(* Logix 5000 project; controller reports 1756-L63 rev 20.15; software revision 20.04; part 32 of 52 *)

        [2].log_data[29].min := 1.0, [2].log_data[29].max := 1.0, [2].log_data[29].total := 3600.0, [2].log_data[29].time := 3600.0, [2].log_data[29].valid := 1, [2].log_data[30].min := 1.0, [2].log_data[30].max := 1.0, [2].log_data[30].total := 3600.0, [2].log_data[30].time := 3600.0, [2].log_data[30].valid := 1, [2].log_data[31].max := 1.0, [2].log_data[31].total := 1162.2471, [2].log_data[31].time := 3600.0, [2].log_data[31].maxminute := 16, [2].log_data[31].valid := 1, [2].log_data[32].max := 1.0, [2].log_data[32].total := 1365.247, [2].log_data[32].time := 3600.0, [2].log_data[32].maxminute := 10, [2].log_data[32].valid := 1, [2].log_data[33].time := 3600.0, [2].log_data[33].valid := 1, [2].log_data[34].time := 3600.0, [2].log_data[34].valid := 1, [2].log_data[35].max := 1.0, [2].log_data[35].total := 1525.747, [2].log_data[35].time := 3600.0, [2].log_data[35].maxminute := 10, [2].log_data[35].valid := 1, [2].log_data[36].max := 1.0, [2].log_data[36].total := 1086.749, [2].log_data[36].time := 3600.0, [2].log_data[36].maxminute := 19, [2].log_data[36].valid := 1, [2].log_data[37].max := 7.628602, [2].log_data[37].total := 3405.06, [2].log_data[37].time := 3600.0, [2].log_data[37].maxminute := 7, [2].log_data[37].valid := 1, [2].log_data[38].time := 3600.0, [2].log_data[38].valid := 1, [2].log_data[39].min := 0.9947063, [2].log_data[39].max := 1.0214411, [2].log_data[39].total := 3607.0884, [2].log_data[39].time := 3600.0, [2].log_data[39].minminute := 23, [2].log_data[39].maxminute := 9, [2].log_data[39].valid := 1, [2].log_data[40].min := 7.538759, [2].log_data[40].max := 7.5879498, [2].log_data[40].total := 27269.645, [2].log_data[40].time := 3600.0, [2].log_data[40].minminute := 15, [2].log_data[40].maxminute := 21, [2].log_data[40].valid := 1, [2].log_data[41].min := 0.046291504, [2].log_data[41].max := 0.07318335, [2].log_data[41].total := 210.1296, [2].log_data[41].time := 3600.0, [2].log_data[41].minminute := 17,
        [2].log_data[41].maxminute := 38, [2].log_data[41].valid := 1, [2].log_data[42].min := 2.2874026, [2].log_data[42].max := 2.2989445, [2].log_data[42].total := 8264.829, [2].log_data[42].time := 3600.0, [2].log_data[42].minminute := 26, [2].log_data[42].maxminute := 48, [2].log_data[42].valid := 1, [2].log_data[43].min := -0.26000214, [2].log_data[43].max := -0.26000214, [2].log_data[43].total := -935.9732, [2].log_data[43].time := 3600.0, [2].log_data[43].valid := 1, [2].log_data[44].min := -0.30000305, [2].log_data[44].max := -0.27999878, [2].log_data[44].total := -1041.974, [2].log_data[44].time := 3600.0, [2].log_data[44].valid := 1, [2].log_data[45].time := 3600.0, [2].log_data[45].valid := 1, [2].log_data[46].time := 3600.0, [2].log_data[46].valid := 1, [2].log_data[47].time := 3600.0, [2].log_data[47].valid := 1, [2].log_data[48].min := 6.583802, [2].log_data[48].max := 6.980899, [2].log_data[48].total := 24245.068, [2].log_data[48].time := 3600.0, [2].log_data[48].minminute := 38, [2].log_data[48].maxminute := 14, [2].log_data[48].valid := 1, [2].log_data[49].min := 6.739631, [2].log_data[49].max := 9.3503065, [2].log_data[49].total := 28682.559, [2].log_data[49].time := 3600.0, [2].log_data[49].minminute := 30, [2].log_data[49].maxminute := 1, [2].log_data[49].valid := 1, [2].log_data[50].min := 2.0478487, [2].log_data[50].max := 2.1506662, [2].log_data[50].total := 7513.924, [2].log_data[50].time := 3600.0, [2].log_data[50].minminute := 59, [2].log_data[50].maxminute := 10, [2].log_data[50].valid := 1, [2].log_data[51].time := 3600.0, [2].log_data[51].valid := 1, [2].log_data[52].min := -4.159996, [2].log_data[52].max := 0.11999512, [2].log_data[52].total := -7228.672, [2].log_data[52].time := 3600.0, [2].log_data[52].minminute := 10, [2].log_data[52].maxminute := 15, [2].log_data[52].valid := 1, [2].log_data[53].min := -3.899994, [2].log_data[53].max := 0.22000122, [2].log_data[53].total := -6730.6216, [2].log_data[53].time := 3600.0, [2].log_data[53].minminute := 10,
        [2].log_data[53].maxminute := 18, [2].log_data[53].valid := 1, [2].log_data[54].max := 0.519, [2].log_data[54].total := 999.3493, [2].log_data[54].time := 3600.0, [2].log_data[54].maxminute := 48, [2].log_data[54].valid := 1, [2].log_data[55].max := 0.534, [2].log_data[55].total := 1035.1941, [2].log_data[55].time := 3600.0, [2].log_data[55].maxminute := 51, [2].log_data[55].valid := 1, [2].log_data[56].min := 0.16024561, [2].log_data[56].max := 0.1607167, [2].log_data[56].total := 577.607, [2].log_data[56].time := 3600.0, [2].log_data[56].minminute := 35, [2].log_data[56].maxminute := 17, [2].log_data[56].valid := 1, [2].log_data[57].min := 0.32045865, [2].log_data[57].max := 0.3224608, [2].log_data[57].total := 1158.1218, [2].log_data[57].time := 3600.0, [2].log_data[57].minminute := 47, [2].log_data[57].maxminute := 30, [2].log_data[57].valid := 1, [2].log_data[58].time := 3600.0, [2].log_data[58].valid := 1, [2].log_data[59].time := 3600.0, [2].log_data[59].valid := 1, [2].log_data[60].valid := 1, [2].log_data[61].valid := 1, [2].log_data[62].valid := 1, [2].log_data[63].valid := 1, [2].log_data[64].valid := 1, [2].log_data[65].valid := 1, [2].log_data[66].valid := 1, [2].log_data[67].valid := 1, [2].log_data[68].valid := 1, [2].log_data[69].valid := 1, [2].log_data[70].valid := 1, [2].log_data[71].valid := 1, [2].log_data[72].valid := 1, [2].log_data[73].valid := 1, [2].log_data[74].valid := 1, [2].log_data[75].valid := 1, [2].log_data[76].valid := 1, [2].log_data[77].valid := 1, [2].log_data[78].valid := 1, [2].log_data[79].valid := 1, [2].log_data[80].valid := 1, [2].log_data[81].valid := 1, [2].log_data[82].valid := 1, [2].log_data[83].valid := 1, [2].log_data[84].valid := 1, [2].log_data[85].valid := 1, [2].log_data[86].valid := 1, [2].log_data[87].valid := 1, [2].log_data[88].valid := 1, [2].log_data[89].valid := 1,
        [2].log_data[90].valid := 1, [2].log_data[91].valid := 1, [2].log_data[92].valid := 1, [2].log_data[93].valid := 1, [2].log_data[94].valid := 1, [2].log_data[95].valid := 1, [2].log_data[96].valid := 1, [2].log_data[97].valid := 1, [2].log_data[98].valid := 1, [2].log_data[99].valid := 1, [2].log_data[100].valid := 1, [2].log_data[101].valid := 1, [2].log_data[102].valid := 1, [2].log_data[103].valid := 1, [2].log_data[104].valid := 1, [2].log_data[105].valid := 1, [2].log_data[106].valid := 1, [2].log_data[107].valid := 1, [2].log_data[108].valid := 1, [2].log_data[109].valid := 1, [2].log_data[110].valid := 1, [2].log_data[111].valid := 1, [2].log_data[112].valid := 1, [2].log_data[113].valid := 1, [2].log_data[114].valid := 1, [2].log_data[115].valid := 1, [2].log_data[116].valid := 1, [2].log_data[117].valid := 1, [2].log_data[118].valid := 1, [2].log_data[119].valid := 1, [2].log_data[120].valid := 1, [2].log_data[121].valid := 1, [2].log_data[122].valid := 1, [2].log_data[123].valid := 1, [2].log_data[124].valid := 1, [2].time.Year := 2023, [2].time.Month := 1, [2].time.Day := 13, [2].time.Hour := 5, [2].time.Minute := 59, [2].time.Second := 59, [3].log_data[0].min := 1.0, [3].log_data[0].max := 1.0, [3].log_data[0].total := 3600.0, [3].log_data[0].time := 3600.0, [3].log_data[0].valid := 1, [3].log_data[1].time := 3600.0, [3].log_data[1].valid := 1, [3].log_data[2].time := 3600.0, [3].log_data[2].valid := 1, [3].log_data[3].time := 3600.0, [3].log_data[3].valid := 1, [3].log_data[4].time := 3600.0, [3].log_data[4].valid := 1, [3].log_data[5].time := 3600.0, [3].log_data[5].valid := 1, [3].log_data[6].time := 3600.0, [3].log_data[6].valid := 1, [3].log_data[7].time := 3600.0, [3].log_data[7].valid := 1,
        [3].log_data[8].max := 1.0, [3].log_data[8].total := 2110.251, [3].log_data[8].time := 3600.0, [3].log_data[8].minminute := 35, [3].log_data[8].valid := 1, [3].log_data[9].max := 1.0, [3].log_data[9].total := 2110.251, [3].log_data[9].time := 3600.0, [3].log_data[9].minminute := 35, [3].log_data[9].valid := 1, [3].log_data[10].min := 1.0, [3].log_data[10].max := 1.0, [3].log_data[10].total := 3600.0, [3].log_data[10].time := 3600.0, [3].log_data[10].valid := 1, [3].log_data[11].time := 3600.0, [3].log_data[11].valid := 1, [3].log_data[12].min := 1.0, [3].log_data[12].max := 1.0, [3].log_data[12].total := 3600.0, [3].log_data[12].time := 3600.0, [3].log_data[12].valid := 1, [3].log_data[13].min := 1.0, [3].log_data[13].max := 1.0, [3].log_data[13].total := 3600.0, [3].log_data[13].time := 3600.0, [3].log_data[13].valid := 1, [3].log_data[14].time := 3600.0, [3].log_data[14].valid := 1, [3].log_data[15].time := 3600.0, [3].log_data[15].valid := 1, [3].log_data[16].time := 3600.0, [3].log_data[16].valid := 1, [3].log_data[17].min := 1.0, [3].log_data[17].max := 1.0, [3].log_data[17].total := 3600.0, [3].log_data[17].time := 3600.0, [3].log_data[17].valid := 1, [3].log_data[18].time := 3600.0, [3].log_data[18].valid := 1, [3].log_data[19].time := 3600.0, [3].log_data[19].valid := 1, [3].log_data[20].time := 3600.0, [3].log_data[20].valid := 1, [3].log_data[21].min := 1.0, [3].log_data[21].max := 1.0, [3].log_data[21].total := 3600.0, [3].log_data[21].time := 3600.0, [3].log_data[21].valid := 1, [3].log_data[22].time := 3600.0, [3].log_data[22].valid := 1, [3].log_data[23].time := 3600.0, [3].log_data[23].valid := 1, [3].log_data[24].time := 3600.0, [3].log_data[24].valid := 1, [3].log_data[25].time := 3600.0, [3].log_data[25].valid := 1, [3].log_data[26].time := 3600.0, [3].log_data[26].valid := 1, [3].log_data[27].time := 3600.0,
        [3].log_data[27].valid := 1, [3].log_data[28].time := 3600.0, [3].log_data[28].valid := 1, [3].log_data[29].min := 1.0, [3].log_data[29].max := 1.0, [3].log_data[29].total := 3600.0, [3].log_data[29].time := 3600.0, [3].log_data[29].valid := 1, [3].log_data[30].min := 1.0, [3].log_data[30].max := 1.0, [3].log_data[30].total := 3600.0, [3].log_data[30].time := 3600.0, [3].log_data[30].valid := 1, [3].log_data[31].max := 1.0, [3].log_data[31].total := 1010.749, [3].log_data[31].time := 3600.0, [3].log_data[31].minminute := 7, [3].log_data[31].valid := 1, [3].log_data[32].max := 1.0, [3].log_data[32].total := 838.749, [3].log_data[32].time := 3600.0, [3].log_data[32].maxminute := 9, [3].log_data[32].valid := 1, [3].log_data[33].time := 3600.0, [3].log_data[33].valid := 1, [3].log_data[34].time := 3600.0, [3].log_data[34].valid := 1, [3].log_data[35].max := 1.0, [3].log_data[35].total := 674.249, [3].log_data[35].time := 3600.0, [3].log_data[35].valid := 1, [3].log_data[36].max := 1.0, [3].log_data[36].total := 1086.498, [3].log_data[36].time := 3600.0, [3].log_data[36].maxminute := 1, [3].log_data[36].valid := 1, [3].log_data[37].time := 3600.0, [3].log_data[37].valid := 1, [3].log_data[38].time := 3600.0, [3].log_data[38].valid := 1, [3].log_data[39].min := 0.99435294, [3].log_data[39].max := 1.0062482, [3].log_data[39].total := 3601.9426, [3].log_data[39].time := 3600.0, [3].log_data[39].minminute := 6, [3].log_data[39].maxminute := 44, [3].log_data[39].valid := 1, [3].log_data[40].min := 7.5588202, [3].log_data[40].max := 7.5808053, [3].log_data[40].total := 27270.088, [3].log_data[40].time := 3600.0, [3].log_data[40].minminute := 56, [3].log_data[40].maxminute := 26, [3].log_data[40].valid := 1, [3].log_data[41].min := 0.041187745, [3].log_data[41].max := 0.071024165, [3].log_data[41].total := 188.56963, [3].log_data[41].time := 3600.0, [3].log_data[41].minminute := 21, [3].log_data[41].maxminute := 43,
        [3].log_data[41].valid := 1, [3].log_data[42].min := 2.2922316, [3].log_data[42].max := 2.3007112, [3].log_data[42].total := 8264.858, [3].log_data[42].time := 3600.0, [3].log_data[42].minminute := 23, [3].log_data[42].maxminute := 24, [3].log_data[42].valid := 1, [3].log_data[43].min := -0.26000214, [3].log_data[43].max := -0.26000214, [3].log_data[43].total := -935.9732, [3].log_data[43].time := 3600.0, [3].log_data[43].valid := 1, [3].log_data[44].min := -0.30000305, [3].log_data[44].max := -0.27999878, [3].log_data[44].total := -1052.0194, [3].log_data[44].time := 3600.0, [3].log_data[44].valid := 1, [3].log_data[45].time := 3600.0, [3].log_data[45].valid := 1, [3].log_data[46].time := 3600.0, [3].log_data[46].valid := 1, [3].log_data[47].time := 3600.0, [3].log_data[47].valid := 1, [3].log_data[48].min := 6.737969, [3].log_data[48].max := 6.778366, [3].log_data[48].total := 24290.475, [3].log_data[48].time := 3600.0, [3].log_data[48].minminute := 40, [3].log_data[48].valid := 1, [3].log_data[49].min := 8.845053, [3].log_data[49].max := 9.3279295, [3].log_data[49].total := 33251.055, [3].log_data[49].time := 3600.0, [3].log_data[49].maxminute := 42, [3].log_data[49].valid := 1, [3].log_data[50].min := 1.9994433, [3].log_data[50].max := 2.1072073, [3].log_data[50].total := 7396.8003, [3].log_data[50].time := 3600.0, [3].log_data[50].minminute := 35, [3].log_data[50].maxminute := 58, [3].log_data[50].valid := 1, [3].log_data[51].time := 3600.0, [3].log_data[51].valid := 1, [3].log_data[52].min := -2.9000015, [3].log_data[52].max := 0.11999512, [3].log_data[52].total := -6534.5815, [3].log_data[52].time := 3600.0, [3].log_data[52].minminute := 19, [3].log_data[52].maxminute := 7, [3].log_data[52].valid := 1, [3].log_data[53].min := -2.4400024, [3].log_data[53].max := 0.19999695, [3].log_data[53].total := -5788.244, [3].log_data[53].time := 3600.0, [3].log_data[53].minminute := 14, [3].log_data[53].valid := 1, [3].log_data[54].max := 0.539, [3].log_data[54].total := 734.8154,
        [3].log_data[54].time := 3600.0, [3].log_data[54].minminute := 7, [3].log_data[54].maxminute := 19, [3].log_data[54].valid := 1, [3].log_data[55].max := 0.5075, [3].log_data[55].total := 697.1523, [3].log_data[55].time := 3600.0, [3].log_data[55].maxminute := 22, [3].log_data[55].valid := 1, [3].log_data[56].min := 0.16032413, [3].log_data[56].max := 0.1607167, [3].log_data[56].total := 577.6799, [3].log_data[56].time := 3600.0, [3].log_data[56].minminute := 9, [3].log_data[56].maxminute := 2, [3].log_data[56].valid := 1, [3].log_data[57].min := 0.32045865, [3].log_data[57].max := 0.3208905, [3].log_data[57].total := 1154.3016, [3].log_data[57].time := 3600.0, [3].log_data[57].minminute := 43, [3].log_data[57].maxminute := 5, [3].log_data[57].valid := 1, [3].log_data[58].time := 3600.0, [3].log_data[58].valid := 1, [3].log_data[59].time := 3600.0, [3].log_data[59].valid := 1, [3].log_data[60].valid := 1, [3].log_data[61].valid := 1, [3].log_data[62].valid := 1, [3].log_data[63].valid := 1, [3].log_data[64].valid := 1, [3].log_data[65].valid := 1, [3].log_data[66].valid := 1, [3].log_data[67].valid := 1, [3].log_data[68].valid := 1, [3].log_data[69].valid := 1, [3].log_data[70].valid := 1, [3].log_data[71].valid := 1, [3].log_data[72].valid := 1, [3].log_data[73].valid := 1, [3].log_data[74].valid := 1, [3].log_data[75].valid := 1, [3].log_data[76].valid := 1, [3].log_data[77].valid := 1, [3].log_data[78].valid := 1, [3].log_data[79].valid := 1, [3].log_data[80].valid := 1, [3].log_data[81].valid := 1, [3].log_data[82].valid := 1, [3].log_data[83].valid := 1, [3].log_data[84].valid := 1, [3].log_data[85].valid := 1, [3].log_data[86].valid := 1, [3].log_data[87].valid := 1, [3].log_data[88].valid := 1, [3].log_data[89].valid := 1, [3].log_data[90].valid := 1, [3].log_data[91].valid := 1, [3].log_data[92].valid := 1,
        [3].log_data[93].valid := 1, [3].log_data[94].valid := 1, [3].log_data[95].valid := 1, [3].log_data[96].valid := 1, [3].log_data[97].valid := 1, [3].log_data[98].valid := 1, [3].log_data[99].valid := 1, [3].log_data[100].valid := 1, [3].log_data[101].valid := 1, [3].log_data[102].valid := 1, [3].log_data[103].valid := 1, [3].log_data[104].valid := 1, [3].log_data[105].valid := 1, [3].log_data[106].valid := 1, [3].log_data[107].valid := 1, [3].log_data[108].valid := 1, [3].log_data[109].valid := 1, [3].log_data[110].valid := 1, [3].log_data[111].valid := 1, [3].log_data[112].valid := 1, [3].log_data[113].valid := 1, [3].log_data[114].valid := 1, [3].log_data[115].valid := 1, [3].log_data[116].valid := 1, [3].log_data[117].valid := 1, [3].log_data[118].valid := 1, [3].log_data[119].valid := 1, [3].log_data[120].valid := 1, [3].log_data[121].valid := 1, [3].log_data[122].valid := 1, [3].log_data[123].valid := 1, [3].log_data[124].valid := 1, [3].time.Year := 2023, [3].time.Month := 1, [3].time.Day := 13, [3].time.Hour := 6, [3].time.Minute := 59, [3].time.Second := 59, [4].log_data[0].min := 1.0, [4].log_data[0].max := 1.0, [4].log_data[0].total := 3600.0, [4].log_data[0].time := 3600.0, [4].log_data[0].valid := 1, [4].log_data[1].time := 3600.0, [4].log_data[1].valid := 1, [4].log_data[2].time := 3600.0, [4].log_data[2].valid := 1, [4].log_data[3].time := 3600.0, [4].log_data[3].valid := 1, [4].log_data[4].time := 3600.0, [4].log_data[4].valid := 1, [4].log_data[5].time := 3600.0, [4].log_data[5].valid := 1, [4].log_data[6].time := 3600.0, [4].log_data[6].valid := 1, [4].log_data[7].time := 3600.0, [4].log_data[7].valid := 1, [4].log_data[8].time := 3600.0, [4].log_data[8].valid := 1, [4].log_data[9].time := 3600.0,
        [4].log_data[9].valid := 1, [4].log_data[10].min := 1.0, [4].log_data[10].max := 1.0, [4].log_data[10].total := 3600.0, [4].log_data[10].time := 3600.0, [4].log_data[10].valid := 1, [4].log_data[11].time := 3600.0, [4].log_data[11].valid := 1, [4].log_data[12].min := 1.0, [4].log_data[12].max := 1.0, [4].log_data[12].total := 3600.0, [4].log_data[12].time := 3600.0, [4].log_data[12].valid := 1, [4].log_data[13].min := 1.0, [4].log_data[13].max := 1.0, [4].log_data[13].total := 3600.0, [4].log_data[13].time := 3600.0, [4].log_data[13].valid := 1, [4].log_data[14].time := 3600.0, [4].log_data[14].valid := 1, [4].log_data[15].time := 3600.0, [4].log_data[15].valid := 1, [4].log_data[16].time := 3600.0, [4].log_data[16].valid := 1, [4].log_data[17].min := 1.0, [4].log_data[17].max := 1.0, [4].log_data[17].total := 3600.0, [4].log_data[17].time := 3600.0, [4].log_data[17].valid := 1, [4].log_data[18].time := 3600.0, [4].log_data[18].valid := 1, [4].log_data[19].time := 3600.0, [4].log_data[19].valid := 1, [4].log_data[20].time := 3600.0, [4].log_data[20].valid := 1, [4].log_data[21].min := 1.0, [4].log_data[21].max := 1.0, [4].log_data[21].total := 3600.0, [4].log_data[21].time := 3600.0, [4].log_data[21].valid := 1, [4].log_data[22].time := 3600.0, [4].log_data[22].valid := 1, [4].log_data[23].time := 3600.0, [4].log_data[23].valid := 1, [4].log_data[24].time := 3600.0, [4].log_data[24].valid := 1, [4].log_data[25].time := 3600.0, [4].log_data[25].valid := 1, [4].log_data[26].time := 3600.0, [4].log_data[26].valid := 1, [4].log_data[27].time := 3600.0, [4].log_data[27].valid := 1, [4].log_data[28].time := 3600.0, [4].log_data[28].valid := 1, [4].log_data[29].min := 1.0, [4].log_data[29].max := 1.0, [4].log_data[29].total := 3600.0, [4].log_data[29].time := 3600.0, [4].log_data[29].valid := 1, [4].log_data[30].min := 1.0,
        [4].log_data[30].max := 1.0, [4].log_data[30].total := 3600.0, [4].log_data[30].time := 3600.0, [4].log_data[30].valid := 1, [4].log_data[31].time := 3600.0, [4].log_data[31].valid := 1, [4].log_data[32].time := 3600.0, [4].log_data[32].valid := 1, [4].log_data[33].time := 3600.0, [4].log_data[33].valid := 1, [4].log_data[34].time := 3600.0, [4].log_data[34].valid := 1, [4].log_data[35].time := 3600.0, [4].log_data[35].valid := 1, [4].log_data[36].time := 3600.0, [4].log_data[36].valid := 1, [4].log_data[37].time := 3600.0, [4].log_data[37].valid := 1, [4].log_data[38].time := 3600.0, [4].log_data[38].valid := 1, [4].log_data[39].min := 0.99423516, [4].log_data[39].max := 1.0055416, [4].log_data[39].total := 3602.0474, [4].log_data[39].time := 3600.0, [4].log_data[39].minminute := 13, [4].log_data[39].maxminute := 34, [4].log_data[39].valid := 1, [4].log_data[40].min := 7.5442557, [4].log_data[40].max := 7.5989423, [4].log_data[40].total := 27264.574, [4].log_data[40].time := 3600.0, [4].log_data[40].minminute := 22, [4].log_data[40].maxminute := 4, [4].log_data[40].valid := 1, [4].log_data[41].min := 0.0402063, [4].log_data[41].max := 0.07514624, [4].log_data[41].total := 193.19824, [4].log_data[41].time := 3600.0, [4].log_data[41].minminute := 58, [4].log_data[41].maxminute := 6, [4].log_data[41].valid := 1, [4].log_data[42].min := 2.2928205, [4].log_data[42].max := 2.298827, [4].log_data[42].total := 8264.684, [4].log_data[42].time := 3600.0, [4].log_data[42].minminute := 17, [4].log_data[42].maxminute := 44, [4].log_data[42].valid := 1, [4].log_data[43].min := -0.26000214, [4].log_data[43].max := -0.26000214, [4].log_data[43].total := -935.9732, [4].log_data[43].time := 3600.0, [4].log_data[43].valid := 1, [4].log_data[44].min := -0.30000305, [4].log_data[44].max := -0.27999878, [4].log_data[44].total := -1033.2828, [4].log_data[44].time := 3600.0, [4].log_data[44].valid := 1, [4].log_data[45].time := 3600.0, [4].log_data[45].valid := 1,
        [4].log_data[46].time := 3600.0, [4].log_data[46].valid := 1, [4].log_data[47].time := 3600.0, [4].log_data[47].valid := 1, [4].log_data[48].min := 6.740717, [4].log_data[48].max := 6.752809, [4].log_data[48].total := 24294.328, [4].log_data[48].time := 3600.0, [4].log_data[48].maxminute := 46, [4].log_data[48].valid := 1, [4].log_data[49].min := 9.282979, [4].log_data[49].max := 9.357571, [4].log_data[49].total := 33554.664, [4].log_data[49].time := 3600.0, [4].log_data[49].minminute := 3, [4].log_data[49].maxminute := 59, [4].log_data[49].valid := 1, [4].log_data[50].min := 2.1007297, [4].log_data[50].max := 2.111447, [4].log_data[50].total := 7586.518, [4].log_data[50].time := 3600.0, [4].log_data[50].minminute := 1, [4].log_data[50].maxminute := 28, [4].log_data[50].valid := 1, [4].log_data[51].time := 3600.0, [4].log_data[51].valid := 1, [4].log_data[52].min := -1.6200027, [4].log_data[52].max := -1.4400024, [4].log_data[52].total := -5511.6133, [4].log_data[52].time := 3600.0, [4].log_data[52].minminute := 37, [4].log_data[52].maxminute := 2, [4].log_data[52].valid := 1, [4].log_data[53].min := -1.5200043, [4].log_data[53].max := -1.340004, [4].log_data[53].total := -5191.9697, [4].log_data[53].time := 3600.0, [4].log_data[53].minminute := 27, [4].log_data[53].maxminute := 3, [4].log_data[53].valid := 1, [4].log_data[54].time := 3600.0, [4].log_data[54].valid := 1, [4].log_data[55].time := 3600.0, [4].log_data[55].valid := 1, [4].log_data[56].min := 0.16028486, [4].log_data[56].max := 0.16067745, [4].log_data[56].total := 577.60114, [4].log_data[56].time := 3600.0, [4].log_data[56].minminute := 3, [4].log_data[56].maxminute := 20, [4].log_data[56].valid := 1, [4].log_data[57].min := 0.32045865, [4].log_data[57].max := 0.32092974, [4].log_data[57].total := 1154.3279, [4].log_data[57].time := 3600.0, [4].log_data[57].minminute := 14, [4].log_data[57].maxminute := 51, [4].log_data[57].valid := 1, [4].log_data[58].time := 3600.0, [4].log_data[58].valid := 1,
        [4].log_data[59].time := 3600.0, [4].log_data[59].valid := 1, [4].log_data[60].valid := 1, [4].log_data[61].valid := 1, [4].log_data[62].valid := 1, [4].log_data[63].valid := 1, [4].log_data[64].valid := 1, [4].log_data[65].valid := 1, [4].log_data[66].valid := 1, [4].log_data[67].valid := 1, [4].log_data[68].valid := 1, [4].log_data[69].valid := 1, [4].log_data[70].valid := 1, [4].log_data[71].valid := 1, [4].log_data[72].valid := 1, [4].log_data[73].valid := 1, [4].log_data[74].valid := 1, [4].log_data[75].valid := 1, [4].log_data[76].valid := 1, [4].log_data[77].valid := 1, [4].log_data[78].valid := 1, [4].log_data[79].valid := 1, [4].log_data[80].valid := 1, [4].log_data[81].valid := 1, [4].log_data[82].valid := 1, [4].log_data[83].valid := 1, [4].log_data[84].valid := 1, [4].log_data[85].valid := 1, [4].log_data[86].valid := 1, [4].log_data[87].valid := 1, [4].log_data[88].valid := 1, [4].log_data[89].valid := 1, [4].log_data[90].valid := 1, [4].log_data[91].valid := 1, [4].log_data[92].valid := 1, [4].log_data[93].valid := 1, [4].log_data[94].valid := 1, [4].log_data[95].valid := 1, [4].log_data[96].valid := 1, [4].log_data[97].valid := 1, [4].log_data[98].valid := 1, [4].log_data[99].valid := 1, [4].log_data[100].valid := 1, [4].log_data[101].valid := 1, [4].log_data[102].valid := 1, [4].log_data[103].valid := 1, [4].log_data[104].valid := 1, [4].log_data[105].valid := 1, [4].log_data[106].valid := 1, [4].log_data[107].valid := 1, [4].log_data[108].valid := 1, [4].log_data[109].valid := 1, [4].log_data[110].valid := 1, [4].log_data[111].valid := 1, [4].log_data[112].valid := 1, [4].log_data[113].valid := 1, [4].log_data[114].valid := 1, [4].log_data[115].valid := 1, [4].log_data[116].valid := 1, [4].log_data[117].valid := 1,
        [4].log_data[118].valid := 1, [4].log_data[119].valid := 1, [4].log_data[120].valid := 1, [4].log_data[121].valid := 1, [4].log_data[122].valid := 1, [4].log_data[123].valid := 1, [4].log_data[124].valid := 1, [4].time.Year := 2023, [4].time.Month := 1, [4].time.Day := 13, [4].time.Hour := 7, [4].time.Minute := 59, [4].time.Second := 59, [5].log_data[0].min := 1.0, [5].log_data[0].max := 1.0, [5].log_data[0].total := 3600.0, [5].log_data[0].time := 3600.0, [5].log_data[0].valid := 1, [5].log_data[1].max := 1.0, [5].log_data[1].total := 575.0, [5].log_data[1].time := 3600.0, [5].log_data[1].maxminute := 33, [5].log_data[1].valid := 1, [5].log_data[2].max := 1.0, [5].log_data[2].total := 571.5, [5].log_data[2].time := 3600.0, [5].log_data[2].maxminute := 33, [5].log_data[2].valid := 1, [5].log_data[3].time := 3600.0, [5].log_data[3].valid := 1, [5].log_data[4].time := 3600.0, [5].log_data[4].valid := 1, [5].log_data[5].max := 1.0, [5].log_data[5].total := 230.0, [5].log_data[5].time := 3600.0, [5].log_data[5].maxminute := 35, [5].log_data[5].valid := 1, [5].log_data[6].time := 3600.0, [5].log_data[6].valid := 1, [5].log_data[7].time := 3600.0, [5].log_data[7].valid := 1, [5].log_data[8].max := 1.0, [5].log_data[8].total := 1354.249, [5].log_data[8].time := 3600.0, [5].log_data[8].maxminute := 37, [5].log_data[8].valid := 1, [5].log_data[9].max := 1.0, [5].log_data[9].total := 1350.749, [5].log_data[9].time := 3600.0, [5].log_data[9].maxminute := 37, [5].log_data[9].valid := 1, [5].log_data[10].min := 1.0, [5].log_data[10].max := 1.0, [5].log_data[10].total := 3600.0, [5].log_data[10].time := 3600.0, [5].log_data[10].valid := 1, [5].log_data[11].time := 3600.0, [5].log_data[11].valid := 1, [5].log_data[12].min := 1.0, [5].log_data[12].max := 1.0,
        [5].log_data[12].total := 3600.0, [5].log_data[12].time := 3600.0, [5].log_data[12].valid := 1, [5].log_data[13].min := 1.0, [5].log_data[13].max := 1.0, [5].log_data[13].total := 3600.0, [5].log_data[13].time := 3600.0, [5].log_data[13].valid := 1, [5].log_data[14].time := 3600.0, [5].log_data[14].valid := 1, [5].log_data[15].time := 3600.0, [5].log_data[15].valid := 1, [5].log_data[16].time := 3600.0, [5].log_data[16].valid := 1, [5].log_data[17].min := 1.0, [5].log_data[17].max := 1.0, [5].log_data[17].total := 3600.0, [5].log_data[17].time := 3600.0, [5].log_data[17].valid := 1, [5].log_data[18].time := 3600.0, [5].log_data[18].valid := 1, [5].log_data[19].time := 3600.0, [5].log_data[19].valid := 1, [5].log_data[20].time := 3600.0, [5].log_data[20].valid := 1, [5].log_data[21].min := 1.0, [5].log_data[21].max := 1.0, [5].log_data[21].total := 3600.0, [5].log_data[21].time := 3600.0, [5].log_data[21].valid := 1, [5].log_data[22].time := 3600.0, [5].log_data[22].valid := 1, [5].log_data[23].time := 3600.0, [5].log_data[23].valid := 1, [5].log_data[24].time := 3600.0, [5].log_data[24].valid := 1, [5].log_data[25].time := 3600.0, [5].log_data[25].valid := 1, [5].log_data[26].time := 3600.0, [5].log_data[26].valid := 1, [5].log_data[27].time := 3600.0, [5].log_data[27].valid := 1, [5].log_data[28].time := 3600.0, [5].log_data[28].valid := 1, [5].log_data[29].min := 1.0, [5].log_data[29].max := 1.0, [5].log_data[29].total := 3600.0, [5].log_data[29].time := 3600.0, [5].log_data[29].valid := 1, [5].log_data[30].min := 1.0, [5].log_data[30].max := 1.0, [5].log_data[30].total := 3600.0, [5].log_data[30].time := 3600.0, [5].log_data[30].valid := 1, [5].log_data[31].max := 1.0, [5].log_data[31].total := 627.498, [5].log_data[31].time := 3600.0, [5].log_data[31].maxminute := 37, [5].log_data[31].valid := 1, [5].log_data[32].max := 1.0,
        [5].log_data[32].total := 543.5, [5].log_data[32].time := 3600.0, [5].log_data[32].maxminute := 43, [5].log_data[32].valid := 1, [5].log_data[33].time := 3600.0, [5].log_data[33].valid := 1, [5].log_data[34].time := 3600.0, [5].log_data[34].valid := 1, [5].log_data[35].max := 1.0, [5].log_data[35].total := 543.249, [5].log_data[35].time := 3600.0, [5].log_data[35].maxminute := 46, [5].log_data[35].valid := 1, [5].log_data[36].max := 1.0, [5].log_data[36].total := 623.998, [5].log_data[36].time := 3600.0, [5].log_data[36].maxminute := 37, [5].log_data[36].valid := 1, [5].log_data[37].max := 7.016958, [5].log_data[37].total := 3500.9973, [5].log_data[37].time := 3600.0, [5].log_data[37].maxminute := 34, [5].log_data[37].valid := 1, [5].log_data[38].time := 3600.0, [5].log_data[38].valid := 1, [5].log_data[39].min := 0.9950596, [5].log_data[39].max := 1.0221478, [5].log_data[39].total := 3609.0261, [5].log_data[39].time := 3600.0, [5].log_data[39].minminute := 4, [5].log_data[39].maxminute := 41, [5].log_data[39].valid := 1, [5].log_data[40].min := 7.5459046, [5].log_data[40].max := 7.590698, [5].log_data[40].total := 27268.496, [5].log_data[40].time := 3600.0, [5].log_data[40].minminute := 59, [5].log_data[40].maxminute := 18, [5].log_data[40].valid := 1, [5].log_data[41].min := 0.030980714, [5].log_data[41].max := 0.058854003, [5].log_data[41].total := 181.6538, [5].log_data[41].time := 3600.0, [5].log_data[41].minminute := 21, [5].log_data[41].maxminute := 15, [5].log_data[41].valid := 1, [5].log_data[42].min := 2.2922316, [5].log_data[42].max := 2.2984736, [5].log_data[42].total := 8264.53, [5].log_data[42].time := 3600.0, [5].log_data[42].minminute := 44, [5].log_data[42].maxminute := 32, [5].log_data[42].valid := 1, [5].log_data[43].min := -0.26000214, [5].log_data[43].max := -0.26000214, [5].log_data[43].total := -935.9732, [5].log_data[43].time := 3600.0, [5].log_data[43].valid := 1, [5].log_data[44].min := -0.30000305, [5].log_data[44].max := -0.27999878,
        [5].log_data[44].total := -1029.0885, [5].log_data[44].time := 3600.0, [5].log_data[44].valid := 1, [5].log_data[45].time := 3600.0, [5].log_data[45].valid := 1, [5].log_data[46].time := 3600.0, [5].log_data[46].valid := 1, [5].log_data[47].time := 3600.0, [5].log_data[47].valid := 1, [5].log_data[48].min := 6.6137557, [5].log_data[48].max := 6.9366555, [5].log_data[48].total := 24325.88, [5].log_data[48].time := 3600.0, [5].log_data[48].minminute := 59, [5].log_data[48].maxminute := 38, [5].log_data[48].valid := 1, [5].log_data[49].min := 6.740613, [5].log_data[49].max := 9.397221, [5].log_data[49].total := 31461.621, [5].log_data[49].time := 3600.0, [5].log_data[49].minminute := 59, [5].log_data[49].maxminute := 24, [5].log_data[49].valid := 1, [5].log_data[50].min := 2.0649261, [5].log_data[50].max := 2.1504307, [5].log_data[50].total := 7575.8022, [5].log_data[50].time := 3600.0, [5].log_data[50].minminute := 41, [5].log_data[50].maxminute := 37, [5].log_data[50].valid := 1, [5].log_data[51].time := 3600.0, [5].log_data[51].valid := 1, [5].log_data[52].min := -4.199997, [5].log_data[52].max := 0.11999512, [5].log_data[52].total := -6420.016, [5].log_data[52].time := 3600.0, [5].log_data[52].minminute := 37, [5].log_data[52].maxminute := 41, [5].log_data[52].valid := 1, [5].log_data[53].min := -3.9399948, [5].log_data[53].max := 0.22000122, [5].log_data[53].total := -5998.357, [5].log_data[53].time := 3600.0, [5].log_data[53].minminute := 37, [5].log_data[53].maxminute := 45, [5].log_data[53].valid := 1, [5].log_data[54].max := 0.51199996, [5].log_data[54].total := 462.47607, [5].log_data[54].time := 3600.0, [5].log_data[54].maxminute := 53, [5].log_data[54].valid := 1, [5].log_data[55].max := 0.5145, [5].log_data[55].total := 460.84094, [5].log_data[55].time := 3600.0, [5].log_data[55].maxminute := 46, [5].log_data[55].valid := 1, [5].log_data[56].min := 0.16016708, [5].log_data[56].max := 0.1607167, [5].log_data[56].total := 577.5164, [5].log_data[56].time := 3600.0,
        [5].log_data[56].minminute := 30, [5].log_data[56].maxminute := 2, [5].log_data[56].valid := 1, [5].log_data[57].min := 0.3204979, [5].log_data[57].max := 0.32092974, [5].log_data[57].total := 1154.4246, [5].log_data[57].time := 3600.0, [5].log_data[57].minminute := 54, [5].log_data[57].maxminute := 15, [5].log_data[57].valid := 1, [5].log_data[58].time := 3600.0, [5].log_data[58].valid := 1, [5].log_data[59].time := 3600.0, [5].log_data[59].valid := 1, [5].log_data[60].valid := 1, [5].log_data[61].valid := 1, [5].log_data[62].valid := 1, [5].log_data[63].valid := 1, [5].log_data[64].valid := 1, [5].log_data[65].valid := 1, [5].log_data[66].valid := 1, [5].log_data[67].valid := 1, [5].log_data[68].valid := 1, [5].log_data[69].valid := 1, [5].log_data[70].valid := 1, [5].log_data[71].valid := 1, [5].log_data[72].valid := 1, [5].log_data[73].valid := 1, [5].log_data[74].valid := 1, [5].log_data[75].valid := 1, [5].log_data[76].valid := 1, [5].log_data[77].valid := 1, [5].log_data[78].valid := 1, [5].log_data[79].valid := 1, [5].log_data[80].valid := 1, [5].log_data[81].valid := 1, [5].log_data[82].valid := 1, [5].log_data[83].valid := 1, [5].log_data[84].valid := 1, [5].log_data[85].valid := 1, [5].log_data[86].valid := 1, [5].log_data[87].valid := 1, [5].log_data[88].valid := 1, [5].log_data[89].valid := 1, [5].log_data[90].valid := 1, [5].log_data[91].valid := 1, [5].log_data[92].valid := 1, [5].log_data[93].valid := 1, [5].log_data[94].valid := 1, [5].log_data[95].valid := 1, [5].log_data[96].valid := 1, [5].log_data[97].valid := 1, [5].log_data[98].valid := 1, [5].log_data[99].valid := 1, [5].log_data[100].valid := 1, [5].log_data[101].valid := 1, [5].log_data[102].valid := 1, [5].log_data[103].valid := 1, [5].log_data[104].valid := 1, [5].log_data[105].valid := 1,
        [5].log_data[106].valid := 1, [5].log_data[107].valid := 1, [5].log_data[108].valid := 1, [5].log_data[109].valid := 1, [5].log_data[110].valid := 1, [5].log_data[111].valid := 1, [5].log_data[112].valid := 1, [5].log_data[113].valid := 1, [5].log_data[114].valid := 1, [5].log_data[115].valid := 1, [5].log_data[116].valid := 1, [5].log_data[117].valid := 1, [5].log_data[118].valid := 1, [5].log_data[119].valid := 1, [5].log_data[120].valid := 1, [5].log_data[121].valid := 1, [5].log_data[122].valid := 1, [5].log_data[123].valid := 1, [5].log_data[124].valid := 1, [5].time.Year := 2023, [5].time.Month := 1, [5].time.Day := 13, [5].time.Hour := 8, [5].time.Minute := 59, [5].time.Second := 59, [6].log_data[0].min := 1.0, [6].log_data[0].max := 1.0, [6].log_data[0].total := 3600.0, [6].log_data[0].time := 3600.0, [6].log_data[0].valid := 1, [6].log_data[1].max := 1.0, [6].log_data[1].total := 275.249, [6].log_data[1].time := 3600.0, [6].log_data[1].maxminute := 55, [6].log_data[1].valid := 1, [6].log_data[2].max := 1.0, [6].log_data[2].total := 271.749, [6].log_data[2].time := 3600.0, [6].log_data[2].maxminute := 55, [6].log_data[2].valid := 1, [6].log_data[3].time := 3600.0, [6].log_data[3].valid := 1, [6].log_data[4].time := 3600.0, [6].log_data[4].valid := 1, [6].log_data[5].max := 1.0, [6].log_data[5].total := 125.5, [6].log_data[5].time := 3600.0, [6].log_data[5].maxminute := 57, [6].log_data[5].valid := 1, [6].log_data[6].time := 3600.0, [6].log_data[6].valid := 1, [6].log_data[7].time := 3600.0, [6].log_data[7].valid := 1, [6].log_data[8].min := 1.0, [6].log_data[8].max := 1.0, [6].log_data[8].total := 3600.0, [6].log_data[8].time := 3600.0, [6].log_data[8].valid := 1, [6].log_data[9].min := 1.0, [6].log_data[9].max := 1.0,
        [6].log_data[9].total := 3600.0, [6].log_data[9].time := 3600.0, [6].log_data[9].valid := 1, [6].log_data[10].min := 1.0, [6].log_data[10].max := 1.0, [6].log_data[10].total := 3600.0, [6].log_data[10].time := 3600.0, [6].log_data[10].valid := 1, [6].log_data[11].time := 3600.0, [6].log_data[11].valid := 1, [6].log_data[12].min := 1.0, [6].log_data[12].max := 1.0, [6].log_data[12].total := 3600.0, [6].log_data[12].time := 3600.0, [6].log_data[12].valid := 1, [6].log_data[13].min := 1.0, [6].log_data[13].max := 1.0, [6].log_data[13].total := 3600.0, [6].log_data[13].time := 3600.0, [6].log_data[13].valid := 1, [6].log_data[14].time := 3600.0, [6].log_data[14].valid := 1, [6].log_data[15].time := 3600.0, [6].log_data[15].valid := 1, [6].log_data[16].time := 3600.0, [6].log_data[16].valid := 1, [6].log_data[17].min := 1.0, [6].log_data[17].max := 1.0, [6].log_data[17].total := 3600.0, [6].log_data[17].time := 3600.0, [6].log_data[17].valid := 1, [6].log_data[18].time := 3600.0, [6].log_data[18].valid := 1, [6].log_data[19].time := 3600.0, [6].log_data[19].valid := 1, [6].log_data[20].time := 3600.0, [6].log_data[20].valid := 1, [6].log_data[21].min := 1.0, [6].log_data[21].max := 1.0, [6].log_data[21].total := 3600.0, [6].log_data[21].time := 3600.0, [6].log_data[21].valid := 1, [6].log_data[22].time := 3600.0, [6].log_data[22].valid := 1, [6].log_data[23].time := 3600.0, [6].log_data[23].valid := 1, [6].log_data[24].time := 3600.0, [6].log_data[24].valid := 1, [6].log_data[25].time := 3600.0, [6].log_data[25].valid := 1, [6].log_data[26].time := 3600.0, [6].log_data[26].valid := 1, [6].log_data[27].time := 3600.0, [6].log_data[27].valid := 1, [6].log_data[28].time := 3600.0, [6].log_data[28].valid := 1, [6].log_data[29].min := 1.0, [6].log_data[29].max := 1.0, [6].log_data[29].total := 3600.0, [6].log_data[29].time := 3600.0,
        [6].log_data[29].valid := 1, [6].log_data[30].min := 1.0, [6].log_data[30].max := 1.0, [6].log_data[30].total := 3600.0, [6].log_data[30].time := 3600.0, [6].log_data[30].valid := 1, [6].log_data[31].max := 1.0, [6].log_data[31].total := 1440.7471, [6].log_data[31].time := 3600.0, [6].log_data[31].minminute := 2, [6].log_data[31].valid := 1, [6].log_data[32].max := 1.0, [6].log_data[32].total := 1629.998, [6].log_data[32].time := 3600.0, [6].log_data[32].maxminute := 4, [6].log_data[32].valid := 1, [6].log_data[33].time := 3600.0, [6].log_data[33].valid := 1, [6].log_data[34].time := 3600.0, [6].log_data[34].valid := 1, [6].log_data[35].max := 1.0, [6].log_data[35].total := 1629.7471, [6].log_data[35].time := 3600.0, [6].log_data[35].maxminute := 7, [6].log_data[35].valid := 1, [6].log_data[36].max := 1.0, [6].log_data[36].total := 1440.7471, [6].log_data[36].time := 3600.0, [6].log_data[36].minminute := 5, [6].log_data[36].valid := 1, [6].log_data[37].max := 7.609758, [6].log_data[37].total := 2055.723, [6].log_data[37].time := 3600.0, [6].log_data[37].maxminute := 57, [6].log_data[37].valid := 1, [6].log_data[38].time := 3600.0, [6].log_data[38].valid := 1, [6].log_data[39].min := 0.99647284, [6].log_data[39].max := 1.0217944, [6].log_data[39].total := 3609.599, [6].log_data[39].time := 3600.0, [6].log_data[39].minminute := 1, [6].log_data[39].maxminute := 58, [6].log_data[39].valid := 1, [6].log_data[40].min := 7.5373855, [6].log_data[40].max := 7.591798, [6].log_data[40].total := 27273.166, [6].log_data[40].time := 3600.0, [6].log_data[40].maxminute := 6, [6].log_data[40].valid := 1, [6].log_data[41].min := 0.039028566, [6].log_data[41].max := 0.072005615, [6].log_data[41].total := 181.46281, [6].log_data[41].time := 3600.0, [6].log_data[41].minminute := 28, [6].log_data[41].maxminute := 36, [6].log_data[41].valid := 1, [6].log_data[42].min := 2.2928205, [6].log_data[42].max := 2.298827, [6].log_data[42].total := 8264.55,
        [6].log_data[42].time := 3600.0, [6].log_data[42].minminute := 2, [6].log_data[42].maxminute := 36, [6].log_data[42].valid := 1, [6].log_data[43].min := -0.27999878, [6].log_data[43].max := -0.26000214, [6].log_data[43].total := -935.9933, [6].log_data[43].time := 3600.0, [6].log_data[43].minminute := 28, [6].log_data[43].valid := 1, [6].log_data[44].min := -0.30000305, [6].log_data[44].max := -0.27999878, [6].log_data[44].total := -1067.1584, [6].log_data[44].time := 3600.0, [6].log_data[44].valid := 1, [6].log_data[45].time := 3600.0, [6].log_data[45].valid := 1, [6].log_data[46].time := 3600.0, [6].log_data[46].valid := 1, [6].log_data[47].time := 3600.0, [6].log_data[47].valid := 1, [6].log_data[48].min := 6.5821533, [6].log_data[48].max := 6.8849916, [6].log_data[48].total := 24246.365, [6].log_data[48].time := 3600.0, [6].log_data[48].minminute := 4, [6].log_data[48].maxminute := 59, [6].log_data[48].valid := 1, [6].log_data[49].min := 6.760046, [6].log_data[49].max := 9.362476, [6].log_data[49].total := 30855.816, [6].log_data[49].time := 3600.0, [6].log_data[49].maxminute := 58, [6].log_data[49].valid := 1, [6].log_data[50].min := 2.0038009, [6].log_data[50].max := 2.0876565, [6].log_data[50].total := 7366.0083, [6].log_data[50].time := 3600.0, [6].log_data[50].minminute := 57, [6].log_data[50].valid := 1, [6].log_data[51].time := 3600.0, [6].log_data[51].valid := 1, [6].log_data[52].min := -3.040001, [6].log_data[52].max := 0.11999512, [6].log_data[52].total := -7493.9536, [6].log_data[52].time := 3600.0, [6].log_data[52].minminute := 14, [6].log_data[52].maxminute := 2, [6].log_data[52].valid := 1, [6].log_data[53].min := -2.4400024, [6].log_data[53].max := 0.27999878, [6].log_data[53].total := -6821.222, [6].log_data[53].time := 3600.0, [6].log_data[53].minminute := 57, [6].log_data[53].maxminute := 6, [6].log_data[53].valid := 1, [6].log_data[54].max := 0.55550003, [6].log_data[54].total := 1217.0961, [6].log_data[54].time := 3600.0, [6].log_data[54].minminute := 2,
        [6].log_data[54].maxminute := 14, [6].log_data[54].valid := 1, [6].log_data[55].max := 0.517, [6].log_data[55].total := 1217.7288, [6].log_data[55].time := 3600.0, [6].log_data[55].minminute := 5, [6].log_data[55].maxminute := 7, [6].log_data[55].valid := 1, [6].log_data[56].min := 0.16016708, [6].log_data[56].max := 0.16067745, [6].log_data[56].total := 577.3738, [6].log_data[56].time := 3600.0, [6].log_data[56].minminute := 5, [6].log_data[56].maxminute := 34, [6].log_data[56].valid := 1, [6].log_data[57].min := 0.3184172, [6].log_data[57].max := 0.3208512, [6].log_data[57].total := 1147.9331, [6].log_data[57].time := 3600.0, [6].log_data[57].minminute := 40, [6].log_data[57].valid := 1, [6].log_data[58].time := 3600.0, [6].log_data[58].valid := 1, [6].log_data[59].time := 3600.0, [6].log_data[59].valid := 1, [6].log_data[60].valid := 1, [6].log_data[61].valid := 1, [6].log_data[62].valid := 1, [6].log_data[63].valid := 1, [6].log_data[64].valid := 1, [6].log_data[65].valid := 1, [6].log_data[66].valid := 1, [6].log_data[67].valid := 1, [6].log_data[68].valid := 1, [6].log_data[69].valid := 1, [6].log_data[70].valid := 1, [6].log_data[71].valid := 1, [6].log_data[72].valid := 1, [6].log_data[73].valid := 1, [6].log_data[74].valid := 1, [6].log_data[75].valid := 1, [6].log_data[76].valid := 1, [6].log_data[77].valid := 1, [6].log_data[78].valid := 1, [6].log_data[79].valid := 1, [6].log_data[80].valid := 1, [6].log_data[81].valid := 1, [6].log_data[82].valid := 1, [6].log_data[83].valid := 1, [6].log_data[84].valid := 1, [6].log_data[85].valid := 1, [6].log_data[86].valid := 1, [6].log_data[87].valid := 1, [6].log_data[88].valid := 1, [6].log_data[89].valid := 1, [6].log_data[90].valid := 1, [6].log_data[91].valid := 1, [6].log_data[92].valid := 1, [6].log_data[93].valid := 1, [6].log_data[94].valid := 1,
        [6].log_data[95].valid := 1, [6].log_data[96].valid := 1, [6].log_data[97].valid := 1, [6].log_data[98].valid := 1, [6].log_data[99].valid := 1, [6].log_data[100].valid := 1, [6].log_data[101].valid := 1, [6].log_data[102].valid := 1, [6].log_data[103].valid := 1, [6].log_data[104].valid := 1, [6].log_data[105].valid := 1, [6].log_data[106].valid := 1, [6].log_data[107].valid := 1, [6].log_data[108].valid := 1, [6].log_data[109].valid := 1, [6].log_data[110].valid := 1, [6].log_data[111].valid := 1, [6].log_data[112].valid := 1, [6].log_data[113].valid := 1, [6].log_data[114].valid := 1, [6].log_data[115].valid := 1, [6].log_data[116].valid := 1, [6].log_data[117].valid := 1, [6].log_data[118].valid := 1, [6].log_data[119].valid := 1, [6].log_data[120].valid := 1, [6].log_data[121].valid := 1, [6].log_data[122].valid := 1, [6].log_data[123].valid := 1, [6].log_data[124].valid := 1, [6].time.Year := 2023, [6].time.Month := 1, [6].time.Day := 13, [6].time.Hour := 9, [6].time.Minute := 59, [6].time.Second := 59, [7].log_data[0].min := 1.0, [7].log_data[0].max := 1.0, [7].log_data[0].total := 3600.0, [7].log_data[0].time := 3600.0, [7].log_data[0].valid := 1, [7].log_data[1].max := 1.0, [7].log_data[1].total := 271.251, [7].log_data[1].time := 3600.0, [7].log_data[1].minminute := 4, [7].log_data[1].valid := 1, [7].log_data[2].max := 1.0, [7].log_data[2].total := 271.251, [7].log_data[2].time := 3600.0, [7].log_data[2].minminute := 4, [7].log_data[2].valid := 1, [7].log_data[3].time := 3600.0, [7].log_data[3].valid := 1, [7].log_data[4].time := 3600.0, [7].log_data[4].valid := 1, [7].log_data[5].max := 1.0, [7].log_data[5].total := 121.0, [7].log_data[5].time := 3600.0, [7].log_data[5].maxminute := 1, [7].log_data[5].valid := 1,
        [7].log_data[6].time := 3600.0, [7].log_data[6].valid := 1, [7].log_data[7].time := 3600.0, [7].log_data[7].valid := 1, [7].log_data[8].max := 1.0, [7].log_data[8].total := 2319.751, [7].log_data[8].time := 3600.0, [7].log_data[8].minminute := 38, [7].log_data[8].valid := 1, [7].log_data[9].max := 1.0, [7].log_data[9].total := 2319.751, [7].log_data[9].time := 3600.0, [7].log_data[9].minminute := 38, [7].log_data[9].valid := 1, [7].log_data[10].min := 1.0, [7].log_data[10].max := 1.0, [7].log_data[10].total := 3600.0, [7].log_data[10].time := 3600.0, [7].log_data[10].valid := 1, [7].log_data[11].time := 3600.0, [7].log_data[11].valid := 1, [7].log_data[12].min := 1.0, [7].log_data[12].max := 1.0, [7].log_data[12].total := 3600.0, [7].log_data[12].time := 3600.0, [7].log_data[12].valid := 1, [7].log_data[13].min := 1.0, [7].log_data[13].max := 1.0, [7].log_data[13].total := 3600.0, [7].log_data[13].time := 3600.0, [7].log_data[13].valid := 1, [7].log_data[14].time := 3600.0, [7].log_data[14].valid := 1, [7].log_data[15].time := 3600.0, [7].log_data[15].valid := 1, [7].log_data[16].time := 3600.0, [7].log_data[16].valid := 1, [7].log_data[17].min := 1.0, [7].log_data[17].max := 1.0, [7].log_data[17].total := 3600.0, [7].log_data[17].time := 3600.0, [7].log_data[17].valid := 1, [7].log_data[18].time := 3600.0, [7].log_data[18].valid := 1, [7].log_data[19].time := 3600.0, [7].log_data[19].valid := 1, [7].log_data[20].time := 3600.0, [7].log_data[20].valid := 1, [7].log_data[21].min := 1.0, [7].log_data[21].max := 1.0, [7].log_data[21].total := 3600.0, [7].log_data[21].time := 3600.0, [7].log_data[21].valid := 1, [7].log_data[22].time := 3600.0, [7].log_data[22].valid := 1, [7].log_data[23].time := 3600.0, [7].log_data[23].valid := 1, [7].log_data[24].time := 3600.0, [7].log_data[24].valid := 1, [7].log_data[25].time := 3600.0,
        [7].log_data[25].valid := 1, [7].log_data[26].time := 3600.0, [7].log_data[26].valid := 1, [7].log_data[27].time := 3600.0, [7].log_data[27].valid := 1, [7].log_data[28].time := 3600.0, [7].log_data[28].valid := 1, [7].log_data[29].min := 1.0, [7].log_data[29].max := 1.0, [7].log_data[29].total := 3600.0, [7].log_data[29].time := 3600.0, [7].log_data[29].valid := 1, [7].log_data[30].min := 1.0, [7].log_data[30].max := 1.0, [7].log_data[30].total := 3600.0, [7].log_data[30].time := 3600.0, [7].log_data[30].valid := 1, [7].log_data[31].max := 1.0, [7].log_data[31].total := 896.0, [7].log_data[31].time := 3600.0, [7].log_data[31].minminute := 5, [7].log_data[31].valid := 1, [7].log_data[32].max := 1.0, [7].log_data[32].total := 1086.498, [7].log_data[32].time := 3600.0, [7].log_data[32].maxminute := 7, [7].log_data[32].valid := 1, [7].log_data[33].max := 1.0, [7].log_data[33].total := 850.249, [7].log_data[33].time := 3600.0, [7].log_data[33].maxminute := 25, [7].log_data[33].valid := 1, [7].log_data[34].max := 1.0, [7].log_data[34].total := 856.751, [7].log_data[34].time := 3600.0, [7].log_data[34].maxminute := 25, [7].log_data[34].valid := 1, [7].log_data[35].max := 1.0, [7].log_data[35].total := 984.49805, [7].log_data[35].time := 3600.0, [7].log_data[35].maxminute := 10, [7].log_data[35].valid := 1, [7].log_data[36].max := 1.0, [7].log_data[36].total := 1074.249, [7].log_data[36].time := 3600.0, [7].log_data[36].minminute := 8, [7].log_data[36].valid := 1, [7].log_data[37].max := 7.4974785, [7].log_data[37].total := 1555.3423, [7].log_data[37].time := 3600.0, [7].log_data[37].minminute := 3, [7].log_data[37].valid := 1, [7].log_data[38].time := 3600.0, [7].log_data[38].valid := 1, [7].log_data[39].min := 0.99435294, [7].log_data[39].max := 1.0213233, [7].log_data[39].total := 3605.7595, [7].log_data[39].time := 3600.0, [7].log_data[39].minminute := 50, [7].log_data[39].maxminute := 1,
        [7].log_data[39].valid := 1, [7].log_data[40].min := 7.5503016, [7].log_data[40].max := 7.5934467, [7].log_data[40].total := 27273.729, [7].log_data[40].time := 3600.0, [7].log_data[40].minminute := 38, [7].log_data[40].maxminute := 44, [7].log_data[40].valid := 1, [7].log_data[41].min := 0.042169187, [7].log_data[41].max := 0.071024165, [7].log_data[41].total := 190.24805, [7].log_data[41].time := 3600.0, [7].log_data[41].minminute := 35, [7].log_data[41].maxminute := 44, [7].log_data[41].valid := 1, [7].log_data[42].min := 2.292467, [7].log_data[42].max := 2.2991803, [7].log_data[42].total := 8264.44, [7].log_data[42].time := 3600.0, [7].log_data[42].minminute := 14, [7].log_data[42].maxminute := 52, [7].log_data[42].valid := 1, [7].log_data[43].min := -0.27999878, [7].log_data[43].max := -0.26000214, [7].log_data[43].total := -936.1723, [7].log_data[43].time := 3600.0, [7].log_data[43].minminute := 32, [7].log_data[43].valid := 1, [7].log_data[44].min := -0.30000305, [7].log_data[44].max := -0.27999878, [7].log_data[44].total := -1072.0834, [7].log_data[44].time := 3600.0, [7].log_data[44].valid := 1, [7].log_data[45].time := 3600.0, [7].log_data[45].valid := 1, [7].log_data[46].time := 3600.0, [7].log_data[46].valid := 1, [7].log_data[47].time := 3600.0, [7].log_data[47].valid := 1, [7].log_data[48].min := 6.578031, [7].log_data[48].max := 6.9325333, [7].log_data[48].total := 24232.69, [7].log_data[48].time := 3600.0, [7].log_data[48].minminute := 26, [7].log_data[48].maxminute := 4, [7].log_data[48].valid := 1, [7].log_data[49].min := 6.6805477, [7].log_data[49].max := 9.022304, [7].log_data[49].total := 28076.045, [7].log_data[49].time := 3600.0, [7].log_data[49].minminute := 22, [7].log_data[49].maxminute := 59, [7].log_data[49].valid := 1, [7].log_data[50].min := 1.9994433, [7].log_data[50].max := 2.1160402, [7].log_data[50].total := 7484.6787, [7].log_data[50].time := 3600.0, [7].log_data[50].minminute := 38, [7].log_data[50].maxminute := 5, [7].log_data[50].valid := 1,
        [7].log_data[51].max := 3.1369998, [7].log_data[51].total := 2655.7993, [7].log_data[51].time := 3600.0, [7].log_data[51].maxminute := 30, [7].log_data[51].valid := 1, [7].log_data[52].min := -2.8600006, [7].log_data[52].max := 0.11999512, [7].log_data[52].total := -6648.9966, [7].log_data[52].time := 3600.0, [7].log_data[52].minminute := 28, [7].log_data[52].maxminute := 5, [7].log_data[52].valid := 1, [7].log_data[53].min := -2.5600052, [7].log_data[53].max := 0.22000122, [7].log_data[53].total := -6370.4414, [7].log_data[53].time := 3600.0, [7].log_data[53].minminute := 31, [7].log_data[53].maxminute := 9, [7].log_data[53].valid := 1, [7].log_data[54].max := 0.523, [7].log_data[54].total := 787.78613, [7].log_data[54].time := 3600.0, [7].log_data[54].minminute := 5, [7].log_data[54].maxminute := 17, [7].log_data[54].valid := 1, [7].log_data[55].max := 0.50949997, [7].log_data[55].total := 817.8937, [7].log_data[55].time := 3600.0, [7].log_data[55].minminute := 8, [7].log_data[55].maxminute := 31, [7].log_data[55].valid := 1, [7].log_data[56].min := 0.16016708, [7].log_data[56].max := 0.16067745, [7].log_data[56].total := 577.4365, [7].log_data[56].time := 3600.0, [7].log_data[56].minminute := 14, [7].log_data[56].maxminute := 13, [7].log_data[56].valid := 1, [7].log_data[57].min := 0.31649354, [7].log_data[57].max := 0.3188491, [7].log_data[57].total := 1143.1768, [7].log_data[57].time := 3600.0, [7].log_data[57].minminute := 49, [7].log_data[57].valid := 1, [7].log_data[58].time := 3600.0, [7].log_data[58].valid := 1, [7].log_data[59].time := 3600.0, [7].log_data[59].valid := 1, [7].log_data[60].valid := 1, [7].log_data[61].valid := 1, [7].log_data[62].valid := 1, [7].log_data[63].valid := 1, [7].log_data[64].valid := 1, [7].log_data[65].valid := 1, [7].log_data[66].valid := 1, [7].log_data[67].valid := 1, [7].log_data[68].valid := 1, [7].log_data[69].valid := 1, [7].log_data[70].valid := 1, [7].log_data[71].valid := 1,
        [7].log_data[72].valid := 1, [7].log_data[73].valid := 1, [7].log_data[74].valid := 1, [7].log_data[75].valid := 1, [7].log_data[76].valid := 1, [7].log_data[77].valid := 1, [7].log_data[78].valid := 1, [7].log_data[79].valid := 1, [7].log_data[80].valid := 1, [7].log_data[81].valid := 1, [7].log_data[82].valid := 1, [7].log_data[83].valid := 1, [7].log_data[84].valid := 1, [7].log_data[85].valid := 1, [7].log_data[86].valid := 1, [7].log_data[87].valid := 1, [7].log_data[88].valid := 1, [7].log_data[89].valid := 1, [7].log_data[90].valid := 1, [7].log_data[91].valid := 1, [7].log_data[92].valid := 1, [7].log_data[93].valid := 1, [7].log_data[94].valid := 1, [7].log_data[95].valid := 1, [7].log_data[96].valid := 1, [7].log_data[97].valid := 1, [7].log_data[98].valid := 1, [7].log_data[99].valid := 1, [7].log_data[100].valid := 1, [7].log_data[101].valid := 1, [7].log_data[102].valid := 1, [7].log_data[103].valid := 1, [7].log_data[104].valid := 1, [7].log_data[105].valid := 1, [7].log_data[106].valid := 1, [7].log_data[107].valid := 1, [7].log_data[108].valid := 1, [7].log_data[109].valid := 1, [7].log_data[110].valid := 1, [7].log_data[111].valid := 1, [7].log_data[112].valid := 1, [7].log_data[113].valid := 1, [7].log_data[114].valid := 1, [7].log_data[115].valid := 1, [7].log_data[116].valid := 1, [7].log_data[117].valid := 1, [7].log_data[118].valid := 1, [7].log_data[119].valid := 1, [7].log_data[120].valid := 1, [7].log_data[121].valid := 1, [7].log_data[122].valid := 1, [7].log_data[123].valid := 1, [7].log_data[124].valid := 1, [7].time.Year := 2023, [7].time.Month := 1, [7].time.Day := 13, [7].time.Hour := 10, [7].time.Minute := 59, [7].time.Second := 59, [8].log_data[0].min := 1.0,
        [8].log_data[0].max := 1.0, [8].log_data[0].total := 3600.0, [8].log_data[0].time := 3600.0, [8].log_data[0].valid := 1, [8].log_data[1].max := 1.0, [8].log_data[1].total := 572.0, [8].log_data[1].time := 3600.0, [8].log_data[1].maxminute := 19, [8].log_data[1].valid := 1, [8].log_data[2].max := 1.0, [8].log_data[2].total := 568.5, [8].log_data[2].time := 3600.0, [8].log_data[2].maxminute := 19, [8].log_data[2].valid := 1, [8].log_data[3].time := 3600.0, [8].log_data[3].valid := 1, [8].log_data[4].time := 3600.0, [8].log_data[4].valid := 1, [8].log_data[5].max := 1.0, [8].log_data[5].total := 240.0, [8].log_data[5].time := 3600.0, [8].log_data[5].maxminute := 21, [8].log_data[5].valid := 1, [8].log_data[6].time := 3600.0, [8].log_data[6].valid := 1, [8].log_data[7].time := 3600.0, [8].log_data[7].valid := 1, [8].log_data[8].max := 1.0, [8].log_data[8].total := 2126.249, [8].log_data[8].time := 3600.0, [8].log_data[8].maxminute := 24, [8].log_data[8].valid := 1, [8].log_data[9].max := 1.0, [8].log_data[9].total := 2122.749, [8].log_data[9].time := 3600.0, [8].log_data[9].maxminute := 24, [8].log_data[9].valid := 1, [8].log_data[10].min := 1.0, [8].log_data[10].max := 1.0, [8].log_data[10].total := 3600.0, [8].log_data[10].time := 3600.0, [8].log_data[10].valid := 1, [8].log_data[11].time := 3600.0, [8].log_data[11].valid := 1, [8].log_data[12].min := 1.0, [8].log_data[12].max := 1.0, [8].log_data[12].total := 3600.0, [8].log_data[12].time := 3600.0, [8].log_data[12].valid := 1, [8].log_data[13].min := 1.0, [8].log_data[13].max := 1.0, [8].log_data[13].total := 3600.0, [8].log_data[13].time := 3600.0, [8].log_data[13].valid := 1, [8].log_data[14].time := 3600.0, [8].log_data[14].valid := 1, [8].log_data[15].time := 3600.0, [8].log_data[15].valid := 1, [8].log_data[16].time := 3600.0, [8].log_data[16].valid := 1,
        [8].log_data[17].min := 1.0, [8].log_data[17].max := 1.0, [8].log_data[17].total := 3600.0, [8].log_data[17].time := 3600.0, [8].log_data[17].valid := 1, [8].log_data[18].time := 3600.0, [8].log_data[18].valid := 1, [8].log_data[19].time := 3600.0, [8].log_data[19].valid := 1, [8].log_data[20].time := 3600.0, [8].log_data[20].valid := 1, [8].log_data[21].min := 1.0, [8].log_data[21].max := 1.0, [8].log_data[21].total := 3600.0, [8].log_data[21].time := 3600.0, [8].log_data[21].valid := 1, [8].log_data[22].time := 3600.0, [8].log_data[22].valid := 1, [8].log_data[23].time := 3600.0, [8].log_data[23].valid := 1, [8].log_data[24].time := 3600.0, [8].log_data[24].valid := 1, [8].log_data[25].time := 3600.0, [8].log_data[25].valid := 1, [8].log_data[26].time := 3600.0, [8].log_data[26].valid := 1, [8].log_data[27].time := 3600.0, [8].log_data[27].valid := 1, [8].log_data[28].time := 3600.0, [8].log_data[28].valid := 1, [8].log_data[29].min := 1.0, [8].log_data[29].max := 1.0, [8].log_data[29].total := 3600.0, [8].log_data[29].time := 3600.0, [8].log_data[29].valid := 1, [8].log_data[30].min := 1.0, [8].log_data[30].max := 1.0, [8].log_data[30].total := 3600.0, [8].log_data[30].time := 3600.0, [8].log_data[30].valid := 1, [8].log_data[31].max := 1.0, [8].log_data[31].total := 1086.498, [8].log_data[31].time := 3600.0, [8].log_data[31].maxminute := 24, [8].log_data[31].valid := 1, [8].log_data[32].max := 1.0, [8].log_data[32].total := 767.99805, [8].log_data[32].time := 3600.0, [8].log_data[32].maxminute := 35, [8].log_data[32].valid := 1, [8].log_data[33].time := 3600.0, [8].log_data[33].valid := 1, [8].log_data[34].time := 3600.0, [8].log_data[34].valid := 1, [8].log_data[35].max := 1.0, [8].log_data[35].total := 1086.498, [8].log_data[35].time := 3600.0, [8].log_data[35].maxminute := 27, [8].log_data[35].valid := 1, [8].log_data[36].max := 1.0,
        [8].log_data[36].total := 676.247, [8].log_data[36].time := 3600.0, [8].log_data[36].maxminute := 24, [8].log_data[36].valid := 1, [8].log_data[37].max := 7.073882, [8].log_data[37].total := 3522.3918, [8].log_data[37].time := 3600.0, [8].log_data[37].maxminute := 21, [8].log_data[37].valid := 1, [8].log_data[38].time := 3600.0, [8].log_data[38].valid := 1, [8].log_data[39].min := 0.99282193, [8].log_data[39].max := 1.0219122, [8].log_data[39].total := 3606.202, [8].log_data[39].time := 3600.0, [8].log_data[39].minminute := 11, [8].log_data[39].maxminute := 22, [8].log_data[39].valid := 1, [8].log_data[40].min := 7.539309, [8].log_data[40].max := 7.600591, [8].log_data[40].total := 27273.223, [8].log_data[40].time := 3600.0, [8].log_data[40].minminute := 15, [8].log_data[40].maxminute := 27, [8].log_data[40].valid := 1, [8].log_data[41].min := 0.045309816, [8].log_data[41].max := 0.078286864, [8].log_data[41].total := 213.89122, [8].log_data[41].time := 3600.0, [8].log_data[41].minminute := 14, [8].log_data[41].maxminute := 27, [8].log_data[41].valid := 1, [8].log_data[42].min := 2.2927027, [8].log_data[42].max := 2.298827, [8].log_data[42].total := 8264.402, [8].log_data[42].time := 3600.0, [8].log_data[42].minminute := 22, [8].log_data[42].maxminute := 30, [8].log_data[42].valid := 1, [8].log_data[43].min := -0.27999878, [8].log_data[43].max := -0.26000214, [8].log_data[43].total := -936.11316, [8].log_data[43].time := 3600.0, [8].log_data[43].valid := 1, [8].log_data[44].min := -0.30000305, [8].log_data[44].max := -0.27999878, [8].log_data[44].total := -1073.2285, [8].log_data[44].time := 3600.0, [8].log_data[44].valid := 1, [8].log_data[45].time := 3600.0, [8].log_data[45].valid := 1, [8].log_data[46].time := 3600.0, [8].log_data[46].valid := 1, [8].log_data[47].time := 3600.0, [8].log_data[47].valid := 1, [8].log_data[48].min := 6.587924, [8].log_data[48].max := 6.996564, [8].log_data[48].total := 24314.635, [8].log_data[48].time := 3600.0, [8].log_data[48].minminute := 54,
        [8].log_data[48].maxminute := 28, [8].log_data[48].valid := 1, [8].log_data[49].min := 6.7783012, [8].log_data[49].max := 9.311441, [8].log_data[49].total := 29129.031, [8].log_data[49].time := 3600.0, [8].log_data[49].minminute := 45, [8].log_data[49].maxminute := 21, [8].log_data[49].valid := 1, [8].log_data[50].min := 2.0549152, [8].log_data[50].max := 2.1505485, [8].log_data[50].total := 7502.178, [8].log_data[50].time := 3600.0, [8].log_data[50].minminute := 59, [8].log_data[50].maxminute := 24, [8].log_data[50].valid := 1, [8].log_data[51].time := 3600.0, [8].log_data[51].valid := 1, [8].log_data[52].min := -4.3600006, [8].log_data[52].max := 0.11999512, [8].log_data[52].total := -6880.8257, [8].log_data[52].time := 3600.0, [8].log_data[52].minminute := 24, [8].log_data[52].maxminute := 33, [8].log_data[52].valid := 1, [8].log_data[53].min := -3.9399948, [8].log_data[53].max := 0.22000122, [8].log_data[53].total := -6201.8916, [8].log_data[53].time := 3600.0, [8].log_data[53].minminute := 24, [8].log_data[53].maxminute := 37, [8].log_data[53].valid := 1, [8].log_data[54].max := 0.532, [8].log_data[54].total := 733.9855, [8].log_data[54].time := 3600.0, [8].log_data[54].maxminute := 45, [8].log_data[54].valid := 1, [8].log_data[55].max := 0.537, [8].log_data[55].total := 695.37305, [8].log_data[55].time := 3600.0, [8].log_data[55].maxminute := 28, [8].log_data[55].valid := 1, [8].log_data[56].min := 0.16016708, [8].log_data[56].max := 0.16067745, [8].log_data[56].total := 577.4176, [8].log_data[56].time := 3600.0, [8].log_data[56].minminute := 46, [8].log_data[56].maxminute := 27, [8].log_data[56].valid := 1, [8].log_data[57].min := 0.31539434, [8].log_data[57].max := 0.31688613, [8].log_data[57].total := 1139.6729, [8].log_data[57].time := 3600.0, [8].log_data[57].minminute := 59, [8].log_data[57].maxminute := 4, [8].log_data[57].valid := 1, [8].log_data[58].time := 3600.0, [8].log_data[58].valid := 1, [8].log_data[59].time := 3600.0, [8].log_data[59].valid := 1,
        [8].log_data[60].valid := 1, [8].log_data[61].valid := 1, [8].log_data[62].valid := 1, [8].log_data[63].valid := 1, [8].log_data[64].valid := 1, [8].log_data[65].valid := 1, [8].log_data[66].valid := 1, [8].log_data[67].valid := 1, [8].log_data[68].valid := 1, [8].log_data[69].valid := 1, [8].log_data[70].valid := 1, [8].log_data[71].valid := 1, [8].log_data[72].valid := 1, [8].log_data[73].valid := 1, [8].log_data[74].valid := 1, [8].log_data[75].valid := 1, [8].log_data[76].valid := 1, [8].log_data[77].valid := 1, [8].log_data[78].valid := 1, [8].log_data[79].valid := 1, [8].log_data[80].valid := 1, [8].log_data[81].valid := 1, [8].log_data[82].valid := 1, [8].log_data[83].valid := 1, [8].log_data[84].valid := 1, [8].log_data[85].valid := 1, [8].log_data[86].valid := 1, [8].log_data[87].valid := 1, [8].log_data[88].valid := 1, [8].log_data[89].valid := 1, [8].log_data[90].valid := 1, [8].log_data[91].valid := 1, [8].log_data[92].valid := 1, [8].log_data[93].valid := 1, [8].log_data[94].valid := 1, [8].log_data[95].valid := 1, [8].log_data[96].valid := 1, [8].log_data[97].valid := 1, [8].log_data[98].valid := 1, [8].log_data[99].valid := 1, [8].log_data[100].valid := 1, [8].log_data[101].valid := 1, [8].log_data[102].valid := 1, [8].log_data[103].valid := 1, [8].log_data[104].valid := 1, [8].log_data[105].valid := 1, [8].log_data[106].valid := 1, [8].log_data[107].valid := 1, [8].log_data[108].valid := 1, [8].log_data[109].valid := 1, [8].log_data[110].valid := 1, [8].log_data[111].valid := 1, [8].log_data[112].valid := 1, [8].log_data[113].valid := 1, [8].log_data[114].valid := 1, [8].log_data[115].valid := 1, [8].log_data[116].valid := 1, [8].log_data[117].valid := 1, [8].log_data[118].valid := 1, [8].log_data[119].valid := 1,
        [8].log_data[120].valid := 1, [8].log_data[121].valid := 1, [8].log_data[122].valid := 1, [8].log_data[123].valid := 1, [8].log_data[124].valid := 1, [8].time.Year := 2023, [8].time.Month := 1, [8].time.Day := 13, [8].time.Hour := 11, [8].time.Minute := 59, [8].time.Second := 59, [9].log_data[0].min := 1.0, [9].log_data[0].max := 1.0, [9].log_data[0].total := 3600.0, [9].log_data[0].time := 3600.0, [9].log_data[0].valid := 1, [9].log_data[1].max := 1.0, [9].log_data[1].total := 540.5, [9].log_data[1].time := 3600.0, [9].log_data[1].maxminute := 41, [9].log_data[1].valid := 1, [9].log_data[2].max := 1.0, [9].log_data[2].total := 537.0, [9].log_data[2].time := 3600.0, [9].log_data[2].maxminute := 41, [9].log_data[2].valid := 1, [9].log_data[3].time := 3600.0, [9].log_data[3].valid := 1, [9].log_data[4].time := 3600.0, [9].log_data[4].valid := 1, [9].log_data[5].max := 1.0, [9].log_data[5].total := 229.0, [9].log_data[5].time := 3600.0, [9].log_data[5].maxminute := 44, [9].log_data[5].valid := 1, [9].log_data[6].time := 3600.0, [9].log_data[6].valid := 1, [9].log_data[7].time := 3600.0, [9].log_data[7].valid := 1, [9].log_data[8].max := 1.0, [9].log_data[8].total := 3188.0, [9].log_data[8].time := 3600.0, [9].log_data[8].minminute := 39, [9].log_data[8].valid := 1, [9].log_data[9].max := 1.0, [9].log_data[9].total := 3184.5, [9].log_data[9].time := 3600.0, [9].log_data[9].minminute := 39, [9].log_data[9].valid := 1, [9].log_data[10].min := 1.0, [9].log_data[10].max := 1.0, [9].log_data[10].total := 3600.0, [9].log_data[10].time := 3600.0, [9].log_data[10].valid := 1, [9].log_data[11].time := 3600.0, [9].log_data[11].valid := 1, [9].log_data[12].min := 1.0, [9].log_data[12].max := 1.0, [9].log_data[12].total := 3600.0, [9].log_data[12].time := 3600.0,
        [9].log_data[12].valid := 1, [9].log_data[13].min := 1.0, [9].log_data[13].max := 1.0, [9].log_data[13].total := 3600.0, [9].log_data[13].time := 3600.0, [9].log_data[13].valid := 1, [9].log_data[14].time := 3600.0, [9].log_data[14].valid := 1, [9].log_data[15].time := 3600.0, [9].log_data[15].valid := 1, [9].log_data[16].time := 3600.0, [9].log_data[16].valid := 1, [9].log_data[17].min := 1.0, [9].log_data[17].max := 1.0, [9].log_data[17].total := 3600.0, [9].log_data[17].time := 3600.0, [9].log_data[17].valid := 1, [9].log_data[18].time := 3600.0, [9].log_data[18].valid := 1, [9].log_data[19].time := 3600.0, [9].log_data[19].valid := 1, [9].log_data[20].time := 3600.0, [9].log_data[20].valid := 1, [9].log_data[21].min := 1.0, [9].log_data[21].max := 1.0, [9].log_data[21].total := 3600.0, [9].log_data[21].time := 3600.0, [9].log_data[21].valid := 1, [9].log_data[22].time := 3600.0, [9].log_data[22].valid := 1, [9].log_data[23].time := 3600.0, [9].log_data[23].valid := 1, [9].log_data[24].time := 3600.0, [9].log_data[24].valid := 1, [9].log_data[25].time := 3600.0, [9].log_data[25].valid := 1, [9].log_data[26].time := 3600.0, [9].log_data[26].valid := 1, [9].log_data[27].time := 3600.0, [9].log_data[27].valid := 1, [9].log_data[28].time := 3600.0, [9].log_data[28].valid := 1, [9].log_data[29].min := 1.0, [9].log_data[29].max := 1.0, [9].log_data[29].total := 3600.0, [9].log_data[29].time := 3600.0, [9].log_data[29].valid := 1, [9].log_data[30].min := 1.0, [9].log_data[30].max := 1.0, [9].log_data[30].total := 3600.0, [9].log_data[30].time := 3600.0, [9].log_data[30].valid := 1, [9].log_data[31].max := 1.0, [9].log_data[31].total := 1547.2471, [9].log_data[31].time := 3600.0, [9].log_data[31].maxminute := 6, [9].log_data[31].valid := 1, [9].log_data[32].max := 1.0, [9].log_data[32].total := 1196.749, [9].log_data[32].time := 3600.0,
        [9].log_data[32].minminute := 5, [9].log_data[32].valid := 1, [9].log_data[33].time := 3600.0, [9].log_data[33].valid := 1, [9].log_data[34].time := 3600.0, [9].log_data[34].valid := 1, [9].log_data[35].max := 1.0, [9].log_data[35].total := 1606.7471, [9].log_data[35].time := 3600.0, [9].log_data[35].maxminute := 10, [9].log_data[35].valid := 1, [9].log_data[36].max := 1.0, [9].log_data[36].total := 1133.2471, [9].log_data[36].time := 3600.0, [9].log_data[36].minminute := 8, [9].log_data[36].valid := 1, [9].log_data[37].max := 7.5759954, [9].log_data[37].total := 3558.4763, [9].log_data[37].time := 3600.0, [9].log_data[37].maxminute := 42, [9].log_data[37].valid := 1, [9].log_data[38].time := 3600.0, [9].log_data[38].valid := 1, [9].log_data[39].min := 0.9936463, [9].log_data[39].max := 1.0229721, [9].log_data[39].total := 3606.6504, [9].log_data[39].time := 3600.0, [9].log_data[39].minminute := 14, [9].log_data[39].maxminute := 48, [9].log_data[39].valid := 1, [9].log_data[40].min := 7.553049, [9].log_data[40].max := 7.59482, [9].log_data[40].total := 27269.057, [9].log_data[40].time := 3600.0, [9].log_data[40].minminute := 59, [9].log_data[40].maxminute := 29, [9].log_data[40].valid := 1, [9].log_data[41].min := 0.043150634, [9].log_data[41].max := 0.05983545, [9].log_data[41].total := 175.35503, [9].log_data[41].time := 3600.0, [9].log_data[41].minminute := 16, [9].log_data[41].valid := 1, [9].log_data[42].min := 2.2922316, [9].log_data[42].max := 2.2990625, [9].log_data[42].total := 8264.247, [9].log_data[42].time := 3600.0, [9].log_data[42].minminute := 24, [9].log_data[42].maxminute := 5, [9].log_data[42].valid := 1, [9].log_data[43].min := -0.27999878, [9].log_data[43].max := -0.26000214, [9].log_data[43].total := -938.10394, [9].log_data[43].time := 3600.0, [9].log_data[43].valid := 1, [9].log_data[44].min := -0.30000305, [9].log_data[44].max := -0.27999878, [9].log_data[44].total := -1079.6809, [9].log_data[44].time := 3600.0, [9].log_data[44].valid := 1,
        [9].log_data[45].time := 3600.0, [9].log_data[45].valid := 1, [9].log_data[46].time := 3600.0, [9].log_data[46].valid := 1, [9].log_data[47].time := 3600.0, [9].log_data[47].valid := 1, [9].log_data[48].min := 6.66542, [9].log_data[48].max := 6.9910674, [9].log_data[48].total := 24406.303, [9].log_data[48].time := 3600.0, [9].log_data[48].maxminute := 50, [9].log_data[48].valid := 1, [9].log_data[49].min := 7.2507744, [9].log_data[49].max := 9.37975, [9].log_data[49].total := 31528.78, [9].log_data[49].time := 3600.0, [9].log_data[49].minminute := 59, [9].log_data[49].maxminute := 44, [9].log_data[49].valid := 1, [9].log_data[50].min := 1.9992077, [9].log_data[50].max := 2.150313, [9].log_data[50].total := 7382.896, [9].log_data[50].time := 3600.0, [9].log_data[50].minminute := 39, [9].log_data[50].maxminute := 46, [9].log_data[50].valid := 1, [9].log_data[51].time := 3600.0, [9].log_data[51].valid := 1, [9].log_data[52].min := -3.9399948, [9].log_data[52].max := 0.11999512, [9].log_data[52].total := -7203.8623, [9].log_data[52].time := 3600.0, [9].log_data[52].minminute := 46, [9].log_data[52].maxminute := 5, [9].log_data[52].valid := 1, [9].log_data[53].min := -3.8600006, [9].log_data[53].max := 0.22000122, [9].log_data[53].total := -6620.528, [9].log_data[53].time := 3600.0, [9].log_data[53].minminute := 46, [9].log_data[53].maxminute := 9, [9].log_data[53].valid := 1, [9].log_data[54].max := 0.531, [9].log_data[54].total := 1086.3938, [9].log_data[54].time := 3600.0, [9].log_data[54].minminute := 5, [9].log_data[54].maxminute := 27, [9].log_data[54].valid := 1, [9].log_data[55].max := 0.539, [9].log_data[55].total := 1084.9948, [9].log_data[55].time := 3600.0, [9].log_data[55].minminute := 8, [9].log_data[55].maxminute := 31, [9].log_data[55].valid := 1, [9].log_data[56].min := 0.16020635, [9].log_data[56].max := 0.16059892, [9].log_data[56].total := 577.3443, [9].log_data[56].time := 3600.0, [9].log_data[56].minminute := 20, [9].log_data[56].maxminute := 1,
        [9].log_data[56].valid := 1, [9].log_data[57].min := 0.3149625, [9].log_data[57].max := 0.31559062, [9].log_data[57].total := 1134.656, [9].log_data[57].time := 3600.0, [9].log_data[57].minminute := 44, [9].log_data[57].valid := 1, [9].log_data[58].time := 3600.0, [9].log_data[58].valid := 1, [9].log_data[59].time := 3600.0, [9].log_data[59].valid := 1, [9].log_data[60].valid := 1, [9].log_data[61].valid := 1, [9].log_data[62].valid := 1, [9].log_data[63].valid := 1, [9].log_data[64].valid := 1, [9].log_data[65].valid := 1, [9].log_data[66].valid := 1, [9].log_data[67].valid := 1, [9].log_data[68].valid := 1, [9].log_data[69].valid := 1, [9].log_data[70].valid := 1, [9].log_data[71].valid := 1, [9].log_data[72].valid := 1, [9].log_data[73].valid := 1, [9].log_data[74].valid := 1, [9].log_data[75].valid := 1, [9].log_data[76].valid := 1, [9].log_data[77].valid := 1, [9].log_data[78].valid := 1, [9].log_data[79].valid := 1, [9].log_data[80].valid := 1, [9].log_data[81].valid := 1, [9].log_data[82].valid := 1, [9].log_data[83].valid := 1, [9].log_data[84].valid := 1, [9].log_data[85].valid := 1, [9].log_data[86].valid := 1, [9].log_data[87].valid := 1, [9].log_data[88].valid := 1, [9].log_data[89].valid := 1, [9].log_data[90].valid := 1, [9].log_data[91].valid := 1, [9].log_data[92].valid := 1, [9].log_data[93].valid := 1, [9].log_data[94].valid := 1, [9].log_data[95].valid := 1, [9].log_data[96].valid := 1, [9].log_data[97].valid := 1, [9].log_data[98].valid := 1, [9].log_data[99].valid := 1, [9].log_data[100].valid := 1, [9].log_data[101].valid := 1, [9].log_data[102].valid := 1, [9].log_data[103].valid := 1, [9].log_data[104].valid := 1, [9].log_data[105].valid := 1, [9].log_data[106].valid := 1, [9].log_data[107].valid := 1, [9].log_data[108].valid := 1,
        [9].log_data[109].valid := 1, [9].log_data[110].valid := 1, [9].log_data[111].valid := 1, [9].log_data[112].valid := 1, [9].log_data[113].valid := 1, [9].log_data[114].valid := 1, [9].log_data[115].valid := 1, [9].log_data[116].valid := 1, [9].log_data[117].valid := 1, [9].log_data[118].valid := 1, [9].log_data[119].valid := 1, [9].log_data[120].valid := 1, [9].log_data[121].valid := 1, [9].log_data[122].valid := 1, [9].log_data[123].valid := 1, [9].log_data[124].valid := 1, [9].time.Year := 2023, [9].time.Month := 1, [9].time.Day := 13, [9].time.Hour := 12, [9].time.Minute := 59, [9].time.Second := 59, [10].log_data[0].min := 1.0, [10].log_data[0].max := 1.0, [10].log_data[0].total := 3599.5, [10].log_data[0].time := 3599.5, [10].log_data[0].valid := 1, [10].log_data[1].max := 1.0, [10].log_data[1].total := 61.5, [10].log_data[1].time := 3599.5, [10].log_data[1].maxminute := 57, [10].log_data[1].valid := 1, [10].log_data[2].max := 1.0, [10].log_data[2].total := 58.0, [10].log_data[2].time := 3599.5, [10].log_data[2].maxminute := 57, [10].log_data[2].valid := 1, [10].log_data[3].time := 3599.5, [10].log_data[3].valid := 1, [10].log_data[4].time := 3599.5, [10].log_data[4].valid := 1, [10].log_data[5].time := 3599.5, [10].log_data[5].valid := 1, [10].log_data[6].time := 3599.5, [10].log_data[6].valid := 1, [10].log_data[7].time := 3599.5, [10].log_data[7].valid := 1, [10].log_data[8].min := 1.0, [10].log_data[8].max := 1.0, [10].log_data[8].total := 3599.5, [10].log_data[8].time := 3599.5, [10].log_data[8].valid := 1, [10].log_data[9].min := 1.0, [10].log_data[9].max := 1.0, [10].log_data[9].total := 3599.5, [10].log_data[9].time := 3599.5, [10].log_data[9].valid := 1, [10].log_data[10].min := 1.0, [10].log_data[10].max := 1.0, [10].log_data[10].total := 3599.5,
        [10].log_data[10].time := 3599.5, [10].log_data[10].valid := 1, [10].log_data[11].time := 3599.5, [10].log_data[11].valid := 1, [10].log_data[12].min := 1.0, [10].log_data[12].max := 1.0, [10].log_data[12].total := 3599.5, [10].log_data[12].time := 3599.5, [10].log_data[12].valid := 1, [10].log_data[13].min := 1.0, [10].log_data[13].max := 1.0, [10].log_data[13].total := 3599.5, [10].log_data[13].time := 3599.5, [10].log_data[13].valid := 1, [10].log_data[14].time := 3599.5, [10].log_data[14].valid := 1, [10].log_data[15].time := 3599.5, [10].log_data[15].valid := 1, [10].log_data[16].time := 3599.5, [10].log_data[16].valid := 1, [10].log_data[17].min := 1.0, [10].log_data[17].max := 1.0, [10].log_data[17].total := 3599.5, [10].log_data[17].time := 3599.5, [10].log_data[17].valid := 1, [10].log_data[18].time := 3599.5, [10].log_data[18].valid := 1, [10].log_data[19].time := 3599.5, [10].log_data[19].valid := 1, [10].log_data[20].time := 3599.5, [10].log_data[20].valid := 1, [10].log_data[21].min := 1.0, [10].log_data[21].max := 1.0, [10].log_data[21].total := 3599.5, [10].log_data[21].time := 3599.5, [10].log_data[21].valid := 1, [10].log_data[22].time := 3599.5, [10].log_data[22].valid := 1, [10].log_data[23].time := 3599.5, [10].log_data[23].valid := 1, [10].log_data[24].time := 3599.5, [10].log_data[24].valid := 1, [10].log_data[25].time := 3599.5, [10].log_data[25].valid := 1, [10].log_data[26].time := 3599.5, [10].log_data[26].valid := 1, [10].log_data[27].time := 3599.5, [10].log_data[27].valid := 1, [10].log_data[28].time := 3599.5, [10].log_data[28].valid := 1, [10].log_data[29].min := 1.0, [10].log_data[29].max := 1.0, [10].log_data[29].total := 3599.5, [10].log_data[29].time := 3599.5, [10].log_data[29].valid := 1, [10].log_data[30].min := 1.0, [10].log_data[30].max := 1.0, [10].log_data[30].total := 3599.5, [10].log_data[30].time := 3599.5, [10].log_data[30].valid := 1,
        [10].log_data[31].max := 1.0, [10].log_data[31].total := 1629.7471, [10].log_data[31].time := 3599.5, [10].log_data[31].maxminute := 6, [10].log_data[31].valid := 1, [10].log_data[32].max := 1.0, [10].log_data[32].total := 1440.749, [10].log_data[32].time := 3599.5, [10].log_data[32].minminute := 4, [10].log_data[32].valid := 1, [10].log_data[33].time := 3599.5, [10].log_data[33].valid := 1, [10].log_data[34].time := 3599.5, [10].log_data[34].valid := 1, [10].log_data[35].max := 1.0, [10].log_data[35].total := 1583.7471, [10].log_data[35].time := 3599.5, [10].log_data[35].maxminute := 9, [10].log_data[35].valid := 1, [10].log_data[36].max := 1.0, [10].log_data[36].total := 1574.498, [10].log_data[36].time := 3599.5, [10].log_data[36].minminute := 8, [10].log_data[36].valid := 1, [10].log_data[37].max := 2.0433266, [10].log_data[37].total := 97.0836, [10].log_data[37].time := 3599.5, [10].log_data[37].maxminute := 57, [10].log_data[37].valid := 1, [10].log_data[38].time := 3599.5, [10].log_data[38].valid := 1, [10].log_data[39].min := 0.99529505, [10].log_data[39].max := 1.008368, [10].log_data[39].total := 3610.3284, [10].log_data[39].time := 3599.5, [10].log_data[39].minminute := 43, [10].log_data[39].maxminute := 59, [10].log_data[39].valid := 1, [10].log_data[40].min := 7.5459046, [10].log_data[40].max := 7.5928965, [10].log_data[40].total := 27262.355, [10].log_data[40].time := 3599.5, [10].log_data[40].minminute := 32, [10].log_data[40].maxminute := 13, [10].log_data[40].valid := 1, [10].log_data[41].min := 0.03412134, [10].log_data[41].max := 0.072987065, [10].log_data[41].total := 180.6271, [10].log_data[41].time := 3599.5, [10].log_data[41].minminute := 43, [10].log_data[41].maxminute := 48, [10].log_data[41].valid := 1, [10].log_data[42].min := 2.2923493, [10].log_data[42].max := 2.2991803, [10].log_data[42].total := 8263.045, [10].log_data[42].time := 3599.5, [10].log_data[42].minminute := 7, [10].log_data[42].maxminute := 26, [10].log_data[42].valid := 1, [10].log_data[43].min := -0.27999878,
        [10].log_data[43].max := -0.26000214, [10].log_data[43].total := -936.2877, [10].log_data[43].time := 3599.5, [10].log_data[43].valid := 1, [10].log_data[44].min := -0.30000305, [10].log_data[44].max := -0.27999878, [10].log_data[44].total := -1078.4253, [10].log_data[44].time := 3599.5, [10].log_data[44].valid := 1, [10].log_data[45].time := 3599.5, [10].log_data[45].valid := 1, [10].log_data[46].time := 3599.5, [10].log_data[46].valid := 1, [10].log_data[47].time := 3599.5, [10].log_data[47].valid := 1, [10].log_data[48].min := 6.586825, [10].log_data[48].max := 6.7984266, [10].log_data[48].total := 24198.63, [10].log_data[48].time := 3599.5, [10].log_data[48].minminute := 15, [10].log_data[48].maxminute := 29, [10].log_data[48].valid := 1, [10].log_data[49].min := 6.809904, [10].log_data[49].max := 9.3503065, [10].log_data[49].total := 29689.723, [10].log_data[49].time := 3599.5, [10].log_data[49].minminute := 9, [10].log_data[49].maxminute := 59, [10].log_data[49].valid := 1, [10].log_data[50].min := 2.0164027, [10].log_data[50].max := 2.0988452, [10].log_data[50].total := 7405.8223, [10].log_data[50].time := 3599.5, [10].log_data[50].minminute := 59, [10].log_data[50].valid := 1, [10].log_data[51].time := 3599.5, [10].log_data[51].valid := 1, [10].log_data[52].min := -3.0200043, [10].log_data[52].max := 0.11999512, [10].log_data[52].total := -7513.5874, [10].log_data[52].time := 3599.5, [10].log_data[52].minminute := 6, [10].log_data[52].maxminute := 4, [10].log_data[52].valid := 1, [10].log_data[53].min := -2.4400024, [10].log_data[53].max := 0.22000122, [10].log_data[53].total := -7134.91, [10].log_data[53].time := 3599.5, [10].log_data[53].minminute := 20, [10].log_data[53].maxminute := 30, [10].log_data[53].valid := 1, [10].log_data[54].max := 0.549, [10].log_data[54].total := 1217.5002, [10].log_data[54].time := 3599.5, [10].log_data[54].minminute := 4, [10].log_data[54].maxminute := 6, [10].log_data[54].valid := 1, [10].log_data[55].max := 0.523, [10].log_data[55].total := 1253.9705, [10].log_data[55].time := 3599.5,
        [10].log_data[55].minminute := 8, [10].log_data[55].maxminute := 51, [10].log_data[55].valid := 1, [10].log_data[56].min := 0.16020635, [10].log_data[56].max := 0.16063818, [10].log_data[56].total := 577.3418, [10].log_data[56].time := 3599.5, [10].log_data[56].minminute := 18, [10].log_data[56].valid := 1, [10].log_data[57].min := 0.3136277, [10].log_data[57].max := 0.3153551, [10].log_data[57].total := 1130.8545, [10].log_data[57].time := 3599.5, [10].log_data[57].minminute := 29, [10].log_data[57].maxminute := 1, [10].log_data[57].valid := 1, [10].log_data[58].time := 3599.5, [10].log_data[58].valid := 1, [10].log_data[59].time := 3599.5, [10].log_data[59].valid := 1, [10].log_data[60].valid := 1, [10].log_data[61].valid := 1, [10].log_data[62].valid := 1, [10].log_data[63].valid := 1, [10].log_data[64].valid := 1, [10].log_data[65].valid := 1, [10].log_data[66].valid := 1, [10].log_data[67].valid := 1, [10].log_data[68].valid := 1, [10].log_data[69].valid := 1, [10].log_data[70].valid := 1, [10].log_data[71].valid := 1, [10].log_data[72].valid := 1, [10].log_data[73].valid := 1, [10].log_data[74].valid := 1, [10].log_data[75].valid := 1, [10].log_data[76].valid := 1, [10].log_data[77].valid := 1, [10].log_data[78].valid := 1, [10].log_data[79].valid := 1, [10].log_data[80].valid := 1, [10].log_data[81].valid := 1, [10].log_data[82].valid := 1, [10].log_data[83].valid := 1, [10].log_data[84].valid := 1, [10].log_data[85].valid := 1, [10].log_data[86].valid := 1, [10].log_data[87].valid := 1, [10].log_data[88].valid := 1, [10].log_data[89].valid := 1, [10].log_data[90].valid := 1, [10].log_data[91].valid := 1, [10].log_data[92].valid := 1, [10].log_data[93].valid := 1, [10].log_data[94].valid := 1, [10].log_data[95].valid := 1, [10].log_data[96].valid := 1, [10].log_data[97].valid := 1, [10].log_data[98].valid := 1, [10].log_data[99].valid := 1,
        [10].log_data[100].valid := 1, [10].log_data[101].valid := 1, [10].log_data[102].valid := 1, [10].log_data[103].valid := 1, [10].log_data[104].valid := 1, [10].log_data[105].valid := 1, [10].log_data[106].valid := 1, [10].log_data[107].valid := 1, [10].log_data[108].valid := 1, [10].log_data[109].valid := 1, [10].log_data[110].valid := 1, [10].log_data[111].valid := 1, [10].log_data[112].valid := 1, [10].log_data[113].valid := 1, [10].log_data[114].valid := 1, [10].log_data[115].valid := 1, [10].log_data[116].valid := 1, [10].log_data[117].valid := 1, [10].log_data[118].valid := 1, [10].log_data[119].valid := 1, [10].log_data[120].valid := 1, [10].log_data[121].valid := 1, [10].log_data[122].valid := 1, [10].log_data[123].valid := 1, [10].log_data[124].valid := 1, [10].time.Year := 2023, [10].time.Month := 1, [10].time.Day := 13, [10].time.Hour := 13, [10].time.Minute := 59, [10].time.Second := 59, [11].log_data[0].min := 1.0, [11].log_data[0].max := 1.0, [11].log_data[0].total := 3600.0, [11].log_data[0].time := 3600.0, [11].log_data[0].valid := 1, [11].log_data[1].max := 1.0, [11].log_data[1].total := 596.249, [11].log_data[1].time := 3600.0, [11].log_data[1].maxminute := 4, [11].log_data[1].valid := 1, [11].log_data[2].max := 1.0, [11].log_data[2].total := 589.249, [11].log_data[2].time := 3600.0, [11].log_data[2].maxminute := 4, [11].log_data[2].valid := 1, [11].log_data[3].time := 3600.0, [11].log_data[3].valid := 1, [11].log_data[4].time := 3600.0, [11].log_data[4].valid := 1, [11].log_data[5].max := 1.0, [11].log_data[5].total := 244.5, [11].log_data[5].time := 3600.0, [11].log_data[5].maxminute := 6, [11].log_data[5].valid := 1, [11].log_data[6].time := 3600.0, [11].log_data[6].valid := 1, [11].log_data[7].time := 3600.0, [11].log_data[7].valid := 1, [11].log_data[8].min := 1.0,
        [11].log_data[8].max := 1.0, [11].log_data[8].total := 3600.0, [11].log_data[8].time := 3600.0, [11].log_data[8].valid := 1, [11].log_data[9].min := 1.0, [11].log_data[9].max := 1.0, [11].log_data[9].total := 3600.0, [11].log_data[9].time := 3600.0, [11].log_data[9].valid := 1, [11].log_data[10].min := 1.0, [11].log_data[10].max := 1.0, [11].log_data[10].total := 3600.0, [11].log_data[10].time := 3600.0, [11].log_data[10].valid := 1, [11].log_data[11].time := 3600.0, [11].log_data[11].valid := 1, [11].log_data[12].min := 1.0, [11].log_data[12].max := 1.0, [11].log_data[12].total := 3600.0, [11].log_data[12].time := 3600.0, [11].log_data[12].valid := 1, [11].log_data[13].min := 1.0, [11].log_data[13].max := 1.0, [11].log_data[13].total := 3600.0, [11].log_data[13].time := 3600.0, [11].log_data[13].valid := 1, [11].log_data[14].time := 3600.0, [11].log_data[14].valid := 1, [11].log_data[15].time := 3600.0, [11].log_data[15].valid := 1, [11].log_data[16].time := 3600.0, [11].log_data[16].valid := 1, [11].log_data[17].min := 1.0, [11].log_data[17].max := 1.0, [11].log_data[17].total := 3600.0, [11].log_data[17].time := 3600.0, [11].log_data[17].valid := 1, [11].log_data[18].time := 3600.0, [11].log_data[18].valid := 1, [11].log_data[19].time := 3600.0, [11].log_data[19].valid := 1, [11].log_data[20].time := 3600.0, [11].log_data[20].valid := 1, [11].log_data[21].min := 1.0, [11].log_data[21].max := 1.0, [11].log_data[21].total := 3600.0, [11].log_data[21].time := 3600.0, [11].log_data[21].valid := 1, [11].log_data[22].time := 3600.0, [11].log_data[22].valid := 1, [11].log_data[23].time := 3600.0, [11].log_data[23].valid := 1, [11].log_data[24].time := 3600.0, [11].log_data[24].valid := 1, [11].log_data[25].time := 3600.0, [11].log_data[25].valid := 1, [11].log_data[26].time := 3600.0, [11].log_data[26].valid := 1, [11].log_data[27].time := 3600.0, [11].log_data[27].valid := 1,
        [11].log_data[28].time := 3600.0, [11].log_data[28].valid := 1, [11].log_data[29].min := 1.0, [11].log_data[29].max := 1.0, [11].log_data[29].total := 3600.0, [11].log_data[29].time := 3600.0, [11].log_data[29].valid := 1, [11].log_data[30].min := 1.0, [11].log_data[30].max := 1.0, [11].log_data[30].total := 3600.0, [11].log_data[30].time := 3600.0, [11].log_data[30].valid := 1, [11].log_data[31].max := 1.0, [11].log_data[31].total := 1591.498, [11].log_data[31].time := 3600.0, [11].log_data[31].maxminute := 9, [11].log_data[31].valid := 1, [11].log_data[32].max := 1.0, [11].log_data[32].total := 1567.5, [11].log_data[32].time := 3600.0, [11].log_data[32].minminute := 8, [11].log_data[32].valid := 1, [11].log_data[33].time := 3600.0, [11].log_data[33].valid := 1, [11].log_data[34].time := 3600.0, [11].log_data[34].valid := 1, [11].log_data[35].max := 1.0, [11].log_data[35].total := 1440.2471, [11].log_data[35].time := 3600.0, [11].log_data[35].valid := 1, [11].log_data[36].max := 1.0, [11].log_data[36].total := 1630.249, [11].log_data[36].time := 3600.0, [11].log_data[36].maxminute := 2, [11].log_data[36].valid := 1, [11].log_data[37].max := 6.9521813, [11].log_data[37].total := 3615.4797, [11].log_data[37].time := 3600.0, [11].log_data[37].maxminute := 5, [11].log_data[37].valid := 1, [11].log_data[38].time := 3600.0, [11].log_data[38].valid := 1, [11].log_data[39].min := 0.99753284, [11].log_data[39].max := 1.0214411, [11].log_data[39].total := 3617.268, [11].log_data[39].time := 3600.0, [11].log_data[39].minminute := 19, [11].log_data[39].maxminute := 7, [11].log_data[39].valid := 1, [11].log_data[40].min := 7.5459046, [11].log_data[40].max := 7.5879498, [11].log_data[40].total := 27270.908, [11].log_data[40].time := 3600.0, [11].log_data[40].minminute := 32, [11].log_data[40].valid := 1, [11].log_data[41].min := 0.036084227, [11].log_data[41].max := 0.07396851, [11].log_data[41].total := 173.53038, [11].log_data[41].time := 3600.0, [11].log_data[41].minminute := 58,
        [11].log_data[41].maxminute := 4, [11].log_data[41].valid := 1, [11].log_data[42].min := 2.292585, [11].log_data[42].max := 2.2989445, [11].log_data[42].total := 8264.187, [11].log_data[42].time := 3600.0, [11].log_data[42].minminute := 59, [11].log_data[42].maxminute := 34, [11].log_data[42].valid := 1, [11].log_data[43].min := -0.27999878, [11].log_data[43].max := -0.26000214, [11].log_data[43].total := -936.6782, [11].log_data[43].time := 3600.0, [11].log_data[43].minminute := 3, [11].log_data[43].valid := 1, [11].log_data[44].min := -0.30000305, [11].log_data[44].max := -0.27999878, [11].log_data[44].total := -1080.066, [11].log_data[44].time := 3600.0, [11].log_data[44].valid := 1, [11].log_data[45].time := 3600.0, [11].log_data[45].valid := 1, [11].log_data[46].time := 3600.0, [11].log_data[46].valid := 1, [11].log_data[47].time := 3600.0, [11].log_data[47].valid := 1, [11].log_data[48].min := 3.5870214, [11].log_data[48].max := 7.130395, [11].log_data[48].total := 23954.744, [11].log_data[48].time := 3600.0, [11].log_data[48].minminute := 19, [11].log_data[48].maxminute := 16, [11].log_data[48].valid := 1, [11].log_data[49].min := 6.7262836, [11].log_data[49].max := 9.39094, [11].log_data[49].total := 28513.625, [11].log_data[49].time := 3600.0, [11].log_data[49].minminute := 32, [11].log_data[49].maxminute := 7, [11].log_data[49].valid := 1, [11].log_data[50].min := 2.0055676, [11].log_data[50].max := 2.1153336, [11].log_data[50].total := 7468.21, [11].log_data[50].time := 3600.0, [11].log_data[50].minminute := 6, [11].log_data[50].maxminute := 14, [11].log_data[50].valid := 1, [11].log_data[51].time := 3600.0, [11].log_data[51].valid := 1, [11].log_data[52].min := -2.9800034, [11].log_data[52].max := 0.11999512, [11].log_data[52].total := -7760.7373, [11].log_data[52].time := 3600.0, [11].log_data[52].minminute := 51, [11].log_data[52].maxminute := 8, [11].log_data[52].valid := 1, [11].log_data[53].min := -2.4800034, [11].log_data[53].max := 0.2599945, [11].log_data[53].total := -7007.413, [11].log_data[53].time := 3600.0,
        [11].log_data[53].minminute := 12, [11].log_data[53].maxminute := 12, [11].log_data[53].valid := 1, [11].log_data[54].max := 0.5565, [11].log_data[54].total := 1254.7542, [11].log_data[54].time := 3600.0, [11].log_data[54].minminute := 8, [11].log_data[54].maxminute := 9, [11].log_data[54].valid := 1, [11].log_data[55].max := 0.5295, [11].log_data[55].total := 1217.6274, [11].log_data[55].time := 3600.0, [11].log_data[55].maxminute := 54, [11].log_data[55].valid := 1, [11].log_data[56].min := 0.16020635, [11].log_data[56].max := 0.16063818, [11].log_data[56].total := 577.46735, [11].log_data[56].time := 3600.0, [11].log_data[56].minminute := 3, [11].log_data[56].maxminute := 6, [11].log_data[56].valid := 1, [11].log_data[57].min := 0.31217515, [11].log_data[57].max := 0.31402028, [11].log_data[57].total := 1126.4764, [11].log_data[57].time := 3600.0, [11].log_data[57].minminute := 37, [11].log_data[57].maxminute := 13, [11].log_data[57].valid := 1, [11].log_data[58].time := 3600.0, [11].log_data[58].valid := 1, [11].log_data[59].time := 3600.0, [11].log_data[59].valid := 1, [11].log_data[60].valid := 1, [11].log_data[61].valid := 1, [11].log_data[62].valid := 1, [11].log_data[63].valid := 1, [11].log_data[64].valid := 1, [11].log_data[65].valid := 1, [11].log_data[66].valid := 1, [11].log_data[67].valid := 1, [11].log_data[68].valid := 1, [11].log_data[69].valid := 1, [11].log_data[70].valid := 1, [11].log_data[71].valid := 1, [11].log_data[72].valid := 1, [11].log_data[73].valid := 1, [11].log_data[74].valid := 1, [11].log_data[75].valid := 1, [11].log_data[76].valid := 1, [11].log_data[77].valid := 1, [11].log_data[78].valid := 1, [11].log_data[79].valid := 1, [11].log_data[80].valid := 1, [11].log_data[81].valid := 1, [11].log_data[82].valid := 1, [11].log_data[83].valid := 1, [11].log_data[84].valid := 1, [11].log_data[85].valid := 1, [11].log_data[86].valid := 1, [11].log_data[87].valid := 1,
        [11].log_data[88].valid := 1, [11].log_data[89].valid := 1, [11].log_data[90].valid := 1, [11].log_data[91].valid := 1, [11].log_data[92].valid := 1, [11].log_data[93].valid := 1, [11].log_data[94].valid := 1, [11].log_data[95].valid := 1, [11].log_data[96].valid := 1, [11].log_data[97].valid := 1, [11].log_data[98].valid := 1, [11].log_data[99].valid := 1, [11].log_data[100].valid := 1, [11].log_data[101].valid := 1, [11].log_data[102].valid := 1, [11].log_data[103].valid := 1, [11].log_data[104].valid := 1, [11].log_data[105].valid := 1, [11].log_data[106].valid := 1, [11].log_data[107].valid := 1, [11].log_data[108].valid := 1, [11].log_data[109].valid := 1, [11].log_data[110].valid := 1, [11].log_data[111].valid := 1, [11].log_data[112].valid := 1, [11].log_data[113].valid := 1, [11].log_data[114].valid := 1, [11].log_data[115].valid := 1, [11].log_data[116].valid := 1, [11].log_data[117].valid := 1, [11].log_data[118].valid := 1, [11].log_data[119].valid := 1, [11].log_data[120].valid := 1, [11].log_data[121].valid := 1, [11].log_data[122].valid := 1, [11].log_data[123].valid := 1, [11].log_data[124].valid := 1, [11].time.Year := 2023, [11].time.Month := 1, [11].time.Day := 13, [11].time.Hour := 14, [11].time.Minute := 59, [11].time.Second := 59, [12].log_data[0].min := 1.0, [12].log_data[0].max := 1.0, [12].log_data[0].total := 3600.0, [12].log_data[0].time := 3600.0, [12].log_data[0].valid := 1, [12].log_data[1].max := 1.0, [12].log_data[1].total := 194.751, [12].log_data[1].time := 3600.0, [12].log_data[1].minminute := 3, [12].log_data[1].valid := 1, [12].log_data[2].max := 1.0, [12].log_data[2].total := 194.751, [12].log_data[2].time := 3600.0, [12].log_data[2].minminute := 3, [12].log_data[2].valid := 1, [12].log_data[3].time := 3600.0, [12].log_data[3].valid := 1,
        [12].log_data[4].time := 3600.0, [12].log_data[4].valid := 1, [12].log_data[5].max := 1.0, [12].log_data[5].total := 90.5, [12].log_data[5].time := 3600.0, [12].log_data[5].maxminute := 1, [12].log_data[5].valid := 1, [12].log_data[6].time := 3600.0, [12].log_data[6].valid := 1, [12].log_data[7].time := 3600.0, [12].log_data[7].valid := 1, [12].log_data[8].min := 1.0, [12].log_data[8].max := 1.0, [12].log_data[8].total := 3600.0, [12].log_data[8].time := 3600.0, [12].log_data[8].valid := 1, [12].log_data[9].min := 1.0, [12].log_data[9].max := 1.0, [12].log_data[9].total := 3600.0, [12].log_data[9].time := 3600.0, [12].log_data[9].valid := 1, [12].log_data[10].min := 1.0, [12].log_data[10].max := 1.0, [12].log_data[10].total := 3600.0, [12].log_data[10].time := 3600.0, [12].log_data[10].valid := 1, [12].log_data[11].time := 3600.0, [12].log_data[11].valid := 1, [12].log_data[12].min := 1.0, [12].log_data[12].max := 1.0, [12].log_data[12].total := 3600.0, [12].log_data[12].time := 3600.0, [12].log_data[12].valid := 1, [12].log_data[13].min := 1.0, [12].log_data[13].max := 1.0, [12].log_data[13].total := 3600.0, [12].log_data[13].time := 3600.0, [12].log_data[13].valid := 1, [12].log_data[14].time := 3600.0, [12].log_data[14].valid := 1, [12].log_data[15].time := 3600.0, [12].log_data[15].valid := 1, [12].log_data[16].time := 3600.0, [12].log_data[16].valid := 1, [12].log_data[17].min := 1.0, [12].log_data[17].max := 1.0, [12].log_data[17].total := 3600.0, [12].log_data[17].time := 3600.0, [12].log_data[17].valid := 1, [12].log_data[18].time := 3600.0, [12].log_data[18].valid := 1, [12].log_data[19].time := 3600.0, [12].log_data[19].valid := 1, [12].log_data[20].time := 3600.0, [12].log_data[20].valid := 1, [12].log_data[21].min := 1.0, [12].log_data[21].max := 1.0, [12].log_data[21].total := 3600.0, [12].log_data[21].time := 3600.0, [12].log_data[21].valid := 1,
        [12].log_data[22].time := 3600.0, [12].log_data[22].valid := 1, [12].log_data[23].time := 3600.0, [12].log_data[23].valid := 1, [12].log_data[24].time := 3600.0, [12].log_data[24].valid := 1, [12].log_data[25].time := 3600.0, [12].log_data[25].valid := 1, [12].log_data[26].time := 3600.0, [12].log_data[26].valid := 1, [12].log_data[27].time := 3600.0, [12].log_data[27].valid := 1, [12].log_data[28].time := 3600.0, [12].log_data[28].valid := 1, [12].log_data[29].min := 1.0, [12].log_data[29].max := 1.0, [12].log_data[29].total := 3600.0, [12].log_data[29].time := 3600.0, [12].log_data[29].valid := 1, [12].log_data[30].min := 1.0, [12].log_data[30].max := 1.0, [12].log_data[30].total := 3600.0, [12].log_data[30].time := 3600.0, [12].log_data[30].valid := 1, [12].log_data[31].max := 1.0, [12].log_data[31].total := 1440.7471, [12].log_data[31].time := 3600.0, [12].log_data[31].valid := 1, [12].log_data[32].max := 1.0, [12].log_data[32].total := 1630.249, [12].log_data[32].time := 3600.0, [12].log_data[32].maxminute := 2, [12].log_data[32].valid := 1, [12].log_data[33].time := 3600.0, [12].log_data[33].valid := 1, [12].log_data[34].time := 3600.0, [12].log_data[34].valid := 1, [12].log_data[35].max := 1.0, [12].log_data[35].total := 1440.498, [12].log_data[35].time := 3600.0, [12].log_data[35].minminute := 3, [12].log_data[35].valid := 1, [12].log_data[36].max := 1.0, [12].log_data[36].total := 1629.7471, [12].log_data[36].time := 3600.0, [12].log_data[36].maxminute := 5, [12].log_data[36].valid := 1, [12].log_data[37].max := 9.07527, [12].log_data[37].total := 1176.3551, [12].log_data[37].time := 3600.0, [12].log_data[37].minminute := 2, [12].log_data[37].valid := 1, [12].log_data[38].time := 3600.0, [12].log_data[38].valid := 1, [12].log_data[39].min := 0.99435294, [12].log_data[39].max := 1.0217944, [12].log_data[39].total := 3606.369, [12].log_data[39].time := 3600.0, [12].log_data[39].minminute := 37, [12].log_data[39].maxminute := 1,
